// TIA Portal V20 export
DATA_BLOCK "ControlNodes"   // DB68
{ DB_Accessible_From_OPC_UA := 'FALSE' }
AUTHOR : ERsystem_FA2_DH. Kim
// stored: DBAccessibleFromOPCUA false, DBAccessibleFromWebserver false, MemoryReserve 100, Namespace Unit1.Em7
   VAR
      em { ExternalAccessible := 'False'; ExternalVisible := 'False'; ExternalWritable := 'False'} : "LAF_typeEmControlNode";
      cm { ExternalAccessible := 'False'; ExternalVisible := 'False'; ExternalWritable := 'False'} : Struct
         interlock : Struct
            sepaClampnCutterAxisX : "LER_typeAxisInterlock";
            sepaClampnCutterAxisZ : "LER_typeAxisInterlock";
            sepaGripperAxisX : "LER_typeAxisInterlock";
            sepaGripperAxisZ : "LER_typeAxisInterlock";
            sepaGripperAxisC : "LER_typeAxisInterlock";
            jrWinderRearAxisY : "LER_typeAxisInterlock";
            jrWinderFrontAxisY : "LER_typeAxisInterlock";
            jrWinderAxisB : "LER_typeAxisInterlock";
            jrPusherAxisZ : "LER_typeAxisInterlock";
            sepaCutterUpDown : "LER_typeTwoWayActInterlock";
            sepaClampTopUpDown : "LER_typeTwoWayActInterlock";
            sepaClampBottomUpDown : "LER_typeTwoWayActInterlock";
            stackGripperOpenClose : "LER_typeTwoWayActInterlock";
            stackGripperFwdBwd : "LER_typeTwoWayActInterlock";
            jrWinderClampTopRearUpDown : "LER_typeTwoWayActInterlock";
            jrWinderClampBtmRearUpDown : "LER_typeTwoWayActInterlock";
            jrWinderClampTopFrontUpDown : "LER_typeTwoWayActInterlock";
            jrWinderClampBtmFrontUpDown : "LER_typeTwoWayActInterlock";
            pusherRollerFwdBwd : "LER_typeTwoWayActInterlock";
         END_STRUCT;
         Command : Struct
            sepaClampnCutterAxisX : "LER_typeAxisCommand";
            sepaClampnCutterAxisZ : "LER_typeAxisCommand";
            sepaGripperAxisX : "LER_typeAxisCommand";
            sepaGripperAxisZ : "LER_typeAxisCommand";
            sepaGripperAxisC : "LER_typeAxisCommand";
            jrWinderRearAxisY : "LER_typeAxisCommand";
            jrWinderFrontAxisY : "LER_typeAxisCommand";
            jrWinderAxisB : "LER_typeAxisCommand";
            jrPusherAxisZ { S7_SetPoint := 'True'} : "LER_typeAxisCommand";
         END_STRUCT;
         softCam : "Unit1.type_emRelations_em7_SoftCam";
         brakeTest : Struct
            sepaClampnCutterAxisZ : "LER_typeBrakeTestEmControlNoeds";
            sepaGripperAxisZ : "LER_typeBrakeTestEmControlNoeds";
            jrPusherAxisZ : "LER_typeBrakeTestEmControlNoeds";
         END_STRUCT;
         calculateCam : Struct
            sepaClampnCutterAxisX : Struct
               execute : Bool;
               done : Bool;
               busy : Bool;
               error : Bool;
               errorID : DWord;
            END_STRUCT;
            sepaClampnCutterAxisZ : Struct
               execute : Bool;
               done : Bool;
               busy : Bool;
               error : Bool;
               errorID : DWord;
            END_STRUCT;
            jrPusherAxisZ : Struct
               execute : Bool;
               done : Bool;
               busy : Bool;
               error : Bool;
               errorID : DWord;
            END_STRUCT;
         END_STRUCT;
         CamIn : Struct
            sepaClampnCutterAxisX : Struct
               execute : Bool := false;
               MasterOffset : LReal := 0.0;
               SlaveOffset : LReal := 0.0;
               MasterScaling : LReal := 1.0;
               SlaveScaling : LReal := 1.0;
               MasterSyncPosition : LReal := 0.0;
               SyncProfileReference : DInt := 2;
               MasterStartDistance : LReal := 0.0;
               Velocity : LReal := -1.0;
               Acceleration : LReal := -1.0;
               Deceleration : LReal := -1.0;
               Jerk : LReal := -1.0;
               ApplicationMode : DInt := 2;
               SyncDirection : DInt := 3;
               StartSync : Bool;
               InSync : Bool;
               Busy : Bool;
               CommandAborted : Bool;
               Error : Bool;
               ErrorId : Word;
               EndOfProfile : Bool;
            END_STRUCT;
            sepaClampnCutterAxisZ : Struct
               execute : Bool := false;
               MasterOffset : LReal := 0.0;
               SlaveOffset : LReal := 0.0;
               MasterScaling : LReal := 1.0;
               SlaveScaling : LReal := 1.0;
               MasterSyncPosition : LReal := 0.0;
               SyncProfileReference : DInt := 2;
               MasterStartDistance : LReal := 0.0;
               Velocity : LReal := -1.0;
               Acceleration : LReal := -1.0;
               Deceleration : LReal := -1.0;
               Jerk : LReal := -1.0;
               ApplicationMode : DInt := 2;
               SyncDirection : DInt := 3;
               StartSync : Bool;
               InSync : Bool;
               Busy : Bool;
               CommandAborted : Bool;
               Error : Bool;
               ErrorId : Word;
               EndOfProfile : Bool;
            END_STRUCT;
            jrPusherAxisZ : Struct
               execute : Bool := false;
               MasterOffset : LReal := 0.0;
               SlaveOffset : LReal := 0.0;
               MasterScaling : LReal := 1.0;
               SlaveScaling : LReal := 1.0;
               MasterSyncPosition : LReal := 0.0;
               SyncProfileReference : DInt := 2;
               MasterStartDistance : LReal := 0.0;
               Velocity : LReal := -1.0;
               Acceleration : LReal := -1.0;
               Deceleration : LReal := -1.0;
               Jerk : LReal := -1.0;
               ApplicationMode : DInt := 2;
               SyncDirection : DInt := 3;
               StartSync : Bool;
               InSync : Bool;
               Busy : Bool;
               CommandAborted : Bool;
               Error : Bool;
               ErrorId : Word;
               EndOfProfile : Bool;
            END_STRUCT;
         END_STRUCT;
         CamUse : Struct
            CamUse : Bool;
         END_STRUCT;
      END_STRUCT;
      sepaClamp : Struct
         jobs : "LAF_typeJobs";
         sequence { S7_SetPoint := 'True'} : "LAF_typeSequence";
         "step" { S7_SetPoint := 'True'} : "LER_typeStep";
         jobInterface : Struct
            homeJob1 { ExternalAccessible := 'False'; ExternalVisible := 'False'; ExternalWritable := 'False'} : "LER_typeJobInterface";
            gripReadyJob2 { ExternalAccessible := 'False'; ExternalVisible := 'False'; ExternalWritable := 'False'; S7_SetPoint := 'True'} : "LER_typeJobInterface";
            clampAndCuttingJob3 { ExternalAccessible := 'False'; ExternalVisible := 'False'; ExternalWritable := 'False'; S7_SetPoint := 'True'} : "LER_typeJobInterface";
            winderMoveJob4 { ExternalAccessible := 'False'; ExternalVisible := 'False'; ExternalWritable := 'False'; S7_SetPoint := 'True'} : "LER_typeJobInterface";
            sepaWindingJob5 { ExternalAccessible := 'False'; ExternalVisible := 'False'; ExternalWritable := 'False'; S7_SetPoint := 'True'} : "LER_typeJobInterface";
            returnJob6 { ExternalAccessible := 'False'; ExternalVisible := 'False'; ExternalWritable := 'False'; S7_SetPoint := 'True'} : "LER_typeJobInterface";
            unloadCamJob10 { S7_SetPoint := 'True'} : "LER_typeJobInterface";
            unloadStopSyncJob11 { S7_SetPoint := 'True'} : "LER_typeJobInterface";
            unloadReturnJob12 { S7_SetPoint := 'True'} : "LER_typeJobInterface";
         END_STRUCT;
         preOperationCheck : Struct
            partNoDetect : Bool;
            partDetect : Bool;
            Bool3 : Bool;
            Bool4 : Bool;
            Bool5 : Bool;
            Bool6 : Bool;
            Bool7 : Bool;
            Bool8 : Bool;
            Bool9 : Bool;
            Bool10 : Bool;
            Bool11 : Bool;
            Bool12 : Bool;
            Bool13 : Bool;
            Bool14 : Bool;
            Bool15 : Bool;
            Bool16 : Bool;
            Bool17 : Bool;
            Bool18 : Bool;
            Bool19 : Bool;
            Bool20 : Bool;
         END_STRUCT;
      END_STRUCT;
      sepaGripper : Struct
         jobs : "LAF_typeJobs";
         sequence { S7_SetPoint := 'True'} : "LAF_typeSequence";
         "step" { S7_SetPoint := 'True'} : "LER_typeStep";
         jobInterface : Struct
            homeJob1 { ExternalAccessible := 'False'; ExternalVisible := 'False'; ExternalWritable := 'False'; S7_SetPoint := 'True'} : "LER_typeJobInterface";
            loadJob2 { ExternalAccessible := 'False'; ExternalVisible := 'False'; ExternalWritable := 'False'; S7_SetPoint := 'True'} : "LER_typeJobInterface";
            unloadJob3 { ExternalAccessible := 'False'; ExternalVisible := 'False'; ExternalWritable := 'False'; S7_SetPoint := 'True'} : "LER_typeJobInterface";
            reLoadJob4 { ExternalAccessible := 'False'; ExternalVisible := 'False'; ExternalWritable := 'False'; S7_SetPoint := 'True'} : "LER_typeJobInterface";
            reUnloadJob5 { ExternalAccessible := 'False'; ExternalVisible := 'False'; ExternalWritable := 'False'; S7_SetPoint := 'True'} : "LER_typeJobInterface";
            LoadToStackTableJob12 { S7_SetPoint := 'True'} : "LER_typeJobInterface";
            UnLoadToJRWinderJob13 { S7_SetPoint := 'True'} : "LER_typeJobInterface";
            LoadToJRWinderJob15 { S7_SetPoint := 'True'} : "LER_typeJobInterface";
            UnLoadToInspectionJob17 { S7_SetPoint := 'True'} : "LER_typeJobInterface";
            ReturnJob18 { S7_SetPoint := 'True'} : "LER_typeJobInterface";
         END_STRUCT;
         preOperationCheck : Struct
            partNoDetect1 : Bool;
            partDetect1 : Bool;
            partNoDetect2 : Bool;
            partDetect2 : Bool;
            partNoDetect1_Cam : Bool;
            partDetect1_Cam : Bool;
            partDetect2_Cam : Bool;
            partNoDetect2_Cam : Bool;
            partDetect3_Cam : Bool;
            partNoDetect3_Cam : Bool;
            Bool11 : Bool;
            Bool12 : Bool;
            Bool13 : Bool;
            Bool14 : Bool;
            Bool15 : Bool;
            Bool16 : Bool;
            Bool17 : Bool;
            Bool18 : Bool;
            Bool19 : Bool;
            Bool20 : Bool;
         END_STRUCT;
      END_STRUCT;
      jellyRollWinder : Struct
         jobs : "LAF_typeJobs";
         sequence { S7_SetPoint := 'True'} : "LAF_typeSequence";
         "step" { S7_SetPoint := 'True'} : "LER_typeStep";
         jobInterface : Struct
            homeJob1 { ExternalAccessible := 'False'; ExternalVisible := 'False'; ExternalWritable := 'False'; S7_SetPoint := 'True'} : "LER_typeJobInterface";
            loadJob2 { ExternalAccessible := 'False'; ExternalVisible := 'False'; ExternalWritable := 'False'; S7_SetPoint := 'True'} : "LER_typeJobInterface";
            winding1Job3 { ExternalAccessible := 'False'; ExternalVisible := 'False'; ExternalWritable := 'False'; S7_SetPoint := 'True'} : "LER_typeJobInterface";
            pusherReadyJob4 { ExternalAccessible := 'False'; ExternalVisible := 'False'; ExternalWritable := 'False'; S7_SetPoint := 'True'} : "LER_typeJobInterface";
            winding2Job5 { ExternalAccessible := 'False'; ExternalVisible := 'False'; ExternalWritable := 'False'; S7_SetPoint := 'True'} : "LER_typeJobInterface";
            unloadJob6 { ExternalAccessible := 'False'; ExternalVisible := 'False'; ExternalWritable := 'False'; S7_SetPoint := 'True'} : "LER_typeJobInterface";
            camWinding1stJob10 { S7_SetPoint := 'True'} : "LER_typeJobInterface";
            camPusherReadyJob11 { S7_SetPoint := 'True'} : "LER_typeJobInterface";
            camCamStartSyncJob12 { S7_SetPoint := 'True'} : "LER_typeJobInterface";
            camWinding2ndJob13 { S7_SetPoint := 'True'} : "LER_typeJobInterface";
            camStopSyncJob14 { S7_SetPoint := 'True'} : "LER_typeJobInterface";
         END_STRUCT;
         preOperationCheck : Struct
            partNoDetect : Bool;
            partDetect : Bool;
            winding1 : Bool;
            pusherReady : Bool;
            winding2 : Bool;
            Bool6 : Bool;
            Bool7 : Bool;
            Bool8 : Bool;
            Bool9 : Bool;
            Bool10 : Bool;
            Bool11 : Bool;
            Bool12 : Bool;
            Bool13 : Bool;
            Bool14 : Bool;
            Bool15 : Bool;
            Bool16 : Bool;
            Bool17 : Bool;
            Bool18 : Bool;
            Bool19 : Bool;
            Bool20 : Bool;
         END_STRUCT;
      END_STRUCT;
      inspectionInterface : Struct
         BA060 : Struct
            null : Bool;
         END_STRUCT;
      END_STRUCT;
      emRelations : Struct
         em4 : Struct
            softCam : "Unit1.type_emRelations_em4_SoftCam";
            cmStatus : Struct
               null : Bool;
            END_STRUCT;
         END_STRUCT;
         em6 : Struct
            softCam : "Unit1.type_emRelations_em6_SoftCam";
            cmStatus : Struct
               GapPadUpDown : "LBC_typeTwoWayActuatorControlNodeMonitoring";
            END_STRUCT;
         END_STRUCT;
      END_STRUCT;
      motionRelations : Struct
         commands : Struct
            unloadGripComplete : Bool;
            unloadClampLockComplete : Bool;
            unloadClampCuttingComplete : Bool;
            unloadJobComplete : Bool;
         END_STRUCT;
         monitoring : Struct
            stackComplete : Bool;
            stackUpComplete : Bool;
            stackUngripComplete : Bool;
            stackGripComplete : Bool;
         END_STRUCT;
         Config : Struct
            Null : Bool;
         END_STRUCT;
      END_STRUCT;
      cmSepaClampDetectSensor { ExternalAccessible := 'False'; ExternalVisible := 'False'; ExternalWritable := 'False'} : "LBC_typeDigitalSignalControlNode";
      cmSepaGripperDetectSensor { ExternalAccessible := 'False'; ExternalVisible := 'False'; ExternalWritable := 'False'} : "LBC_typeDigitalSignalControlNode";
      cmJRWinderDetectSensor { ExternalAccessible := 'False'; ExternalVisible := 'False'; ExternalWritable := 'False'} : "LBC_typeDigitalSignalControlNode";
      cmSepaClampSafetyPinDetectSensor { ExternalAccessible := 'False'; ExternalVisible := 'False'; ExternalWritable := 'False'} : "LBC_typeDigitalSignalControlNode";
      cmSepaGripperSafetyPinDetectSensor { ExternalAccessible := 'False'; ExternalVisible := 'False'; ExternalWritable := 'False'} : "LBC_typeDigitalSignalControlNode";
      cmSepaClampnCutterAxisX { ExternalAccessible := 'False'; ExternalVisible := 'False'; ExternalWritable := 'False'} : "LBC_typeAxis64PosControlNode";
      cmSepaClampnCutterAxisZ { ExternalAccessible := 'False'; ExternalVisible := 'False'; ExternalWritable := 'False'} : "LBC_typeAxis64PosControlNode";
      cmSepaGripperAxisX { ExternalAccessible := 'False'; ExternalVisible := 'False'; ExternalWritable := 'False'} : "LBC_typeAxis64PosControlNode";
      cmSepaGripperAxisZ { ExternalAccessible := 'False'; ExternalVisible := 'False'; ExternalWritable := 'False'} : "LBC_typeAxis64PosControlNode";
      cmSepaGripperAxisC { ExternalAccessible := 'False'; ExternalVisible := 'False'; ExternalWritable := 'False'} : "LBC_typeAxis64PosControlNode";
      cmJRWinderRearAxisY { ExternalAccessible := 'False'; ExternalVisible := 'False'; ExternalWritable := 'False'} : "LBC_typeAxis64PosControlNode";
      cmJRWinderFrontAxisY { ExternalAccessible := 'False'; ExternalVisible := 'False'; ExternalWritable := 'False'} : "LBC_typeAxis64PosControlNode";
      cmJRWinderAxisB { ExternalAccessible := 'False'; ExternalVisible := 'False'; ExternalWritable := 'False'} : "LBC_typeAxis64PosControlNode";
      cmJRPusherAxisZ { ExternalAccessible := 'False'; ExternalVisible := 'False'; ExternalWritable := 'False'} : "LBC_typeAxis64PosControlNode";
      cmSepaCutterUpDown { ExternalAccessible := 'False'; ExternalVisible := 'False'; ExternalWritable := 'False'} : "LBC_typeTwoWayActuatorControlNode";
      cmSepaClampTopUpDown { ExternalAccessible := 'False'; ExternalVisible := 'False'; ExternalWritable := 'False'} : "LBC_typeTwoWayActuatorControlNode";
      cmSepaClampBottomUpDown { ExternalAccessible := 'False'; ExternalVisible := 'False'; ExternalWritable := 'False'} : "LBC_typeTwoWayActuatorControlNode";
      cmStackGripperOpenClose { ExternalAccessible := 'False'; ExternalVisible := 'False'; ExternalWritable := 'False'} : "LBC_typeTwoWayActuatorControlNode";
      cmStackGripperFwdBwd { ExternalAccessible := 'False'; ExternalVisible := 'False'; ExternalWritable := 'False'} : "LBC_typeTwoWayActuatorControlNode";
      cmJRWinderClampTopRearUpDown { ExternalAccessible := 'False'; ExternalVisible := 'False'; ExternalWritable := 'False'} : "LBC_typeTwoWayActuatorControlNode";
      cmJRWinderClampBtmRearUpDown { ExternalAccessible := 'False'; ExternalVisible := 'False'; ExternalWritable := 'False'} : "LBC_typeTwoWayActuatorControlNode";
      cmJRWinderClampTopFrontUpDown { ExternalAccessible := 'False'; ExternalVisible := 'False'; ExternalWritable := 'False'} : "LBC_typeTwoWayActuatorControlNode";
      cmJRWinderClampBtmFrontUpDown { ExternalAccessible := 'False'; ExternalVisible := 'False'; ExternalWritable := 'False'} : "LBC_typeTwoWayActuatorControlNode";
      cmPusherRollerFwdBwd { ExternalAccessible := 'False'; ExternalVisible := 'False'; ExternalWritable := 'False'} : "LBC_typeTwoWayActuatorControlNode";
      cmHotWireCutter { ExternalAccessible := 'False'; ExternalVisible := 'False'; ExternalWritable := 'False'} : "LER_typeHotWireCutterControlNode";
   END_VAR
BEGIN
   em.commands.enable := FALSE;
   em.commands.acknowledge := FALSE;
   em.commands.disableAlarms := FALSE;
   em.commands.activateSimulation := FALSE;
   em.commands.home := FALSE;
   em.commands.moveToInitialPosition := FALSE;
   em.commands.directModeControl.current := 2;
   em.commands.directModeControl.production := FALSE;
   em.commands.directModeControl.maintenance := TRUE;
   em.commands.directModeControl.manual := FALSE;
   em.commands.directModeControl.nomode := FALSE;
   em.commands.directModeControl.sleep := FALSE;
   em.commands.directModeControl.deepsleep := FALSE;
   em.commands.directModeControl.userMode04 := FALSE;
   em.commands.directModeControl.userMode05 := FALSE;
   em.commands.directModeControl.userMode06 := FALSE;
   em.commands.directModeControl.userMode07 := FALSE;
   em.commands.directModeControl.userMode08 := FALSE;
   em.commands.directModeControl.userMode09 := FALSE;
   em.commands.directModeControl.userMode10 := FALSE;
   em.commands.directModeControl.userMode11 := FALSE;
   em.commands.directModeControl.userMode12 := FALSE;
   em.commands.directModeControl.userMode13 := FALSE;
   em.commands.directStateControl.current := 2;
   em.commands.directStateControl.clearing := FALSE;
   em.commands.directStateControl.stopped := TRUE;
   em.commands.directStateControl.starting := FALSE;
   em.commands.directStateControl.idle := FALSE;
   em.commands.directStateControl.suspended := FALSE;
   em.commands.directStateControl.execute := FALSE;
   em.commands.directStateControl.stopping := FALSE;
   em.commands.directStateControl.aborting := FALSE;
   em.commands.directStateControl.aborted := FALSE;
   em.commands.directStateControl.holding := FALSE;
   em.commands.directStateControl.held := FALSE;
   em.commands.directStateControl.unholding := FALSE;
   em.commands.directStateControl.suspending := FALSE;
   em.commands.directStateControl.unsuspending := FALSE;
   em.commands.directStateControl.resetting := FALSE;
   em.commands.directStateControl.completing := FALSE;
   em.commands.directStateControl.complete := FALSE;
   em.status.enabled := FALSE;
   em.status.acknowledgeActive := FALSE;
   em.status.alarmsDisabled := FALSE;
   em.status.simulationActive := FALSE;
   em.status.safetyReleased := TRUE;
   em.status.initialized := FALSE;
   em.status.homed := FALSE;
   em.status.safeState := FALSE;
   em.status.stateComplete := TRUE;
   // sepaClamp."step".action1[101] : Step[101] : JOB[1] Condition
   // sepaClamp."step".action1[110] : Step[110] : Cutter Up
   // sepaClamp."step".action1[120] : Step[120] : Cutter Heater Off
   // sepaClamp."step".action1[130] : Step[130] : Clamp Close
   // sepaClamp."step".action1[180] : Step[180] : Clamp X,Z-Axis Wait Pos
   // sepaClamp."step".action1[190] : Step[190] : Job[1] Step End
   // sepaClamp."step".action1[201] : Step[201] : JOB[2] Condition
   // sepaClamp."step".action1[210] : Step[210] : Clamp X,Z-Axis Load Pos
   // sepaClamp."step".action1[220] : Step[220] : Clamp Open
   // sepaClamp."step".action1[221] : Step[221] : Sepa Clamp → Sepa Gripper [Loading Ready]
   // sepaClamp."step".action1[230] : Step[230] : Clamp Close
   // sepaClamp."step".action1[240] : Step[240] : Cutter Heater On
   // sepaClamp."step".action1[250] : Step[250] : Cutter Down
   // sepaClamp."step".action1[251] : Step[251] : Cutter Up
   // sepaClamp."step".action1[260] : Step[260] : Cutter Heater Off
   // sepaClamp."step".action1[280] : Step[280] : Clamp X,Z-Axis Winding Ready Pos
   // sepaClamp."step".action1[290] : Step[290] : Job[2] Step End
   // sepaClamp."step".action1[301] : Step[301] : JOB[3] Condition
   // sepaClamp."step".action1[310] : Step[310] : Sepa Clamp → JR Winder [Unloading Ready]
   // sepaClamp."step".action1[320] : Step[320] : Clamp X-Axis Winding Move Pos
   // sepaClamp."step".action1[321] : Step[321] : Sepa Clamp → JR Winder [UnClamp Ready]
   // sepaClamp."step".action1[330] : Step[330] : Clamp Open
   // sepaClamp."step".action1[331] : Step[331] : Sepa Clamp → JR Winder [Unloading Done]
   // sepaClamp."step".action1[340] : Step[340] : Clamp Close
   // sepaClamp."step".action1[380] : Step[380] : Clamp X,Z-Axis Wait Pos
   // sepaClamp."step".action1[390] : Step[390] : Job[3] Step End
   // sepaClamp."step".action1[401] : Step[401] : JOB[4] Condition
   // sepaClamp."step".action1[410] : Step[410] : Clamp X-Axis Winder Pos
   // sepaClamp."step".action1[411] : Step[411] : Clamp Z-Axis Winder Pos
   // sepaClamp."step".action1[490] : Step[490] : Job[4] Step End
   // sepaClamp."step".action1[501] : Step[501] : Job[5] Condition
   // sepaClamp."step".action1[510] : Step[510] : CamIn Config
   // sepaClamp."step".action1[511] : Step[511] : Clamp X-Axis CamIn
   // sepaClamp."step".action1[520] : Step[520] : Check Clamp X-Axis WinderDone Pos
   // sepaClamp."step".action1[521] : Step[521] : Clamp X-Axis Halt
   // sepaClamp."step".action1[530] : Step[530] : Clamp Open
   // sepaClamp."step".action1[590] : Step[590] : Job[5] Step End
   // sepaClamp."step".action1[601] : Step[601] : JOB[6] Condition
   // sepaClamp."step".action1[610] : Step[610] : Cutter Up
   // sepaClamp."step".action1[611] : Step[611] : Clamp Close
   // sepaClamp."step".action1[620] : Step[620] : Clamp Z-Axis WaitPos
   // sepaClamp."step".action1[630] : Step[630] : Clamp X-Axis WaitPos
   // sepaClamp."step".action1[690] : Step[690] : Job[6] Step End
   // sepaClamp."step".action1[1001] : Step[1001] : JOB[10] Condition
   // sepaClamp."step".action1[1010] : Step[1010] : Sepa Clamp X/Z Cam Calculate
   // sepaClamp."step".action1[1011] : Step[1011] : Sepa Clamp X/Z CamIn
   // sepaClamp."step".action1[1090] : Step[1090] : Job[10] Step End
   // sepaClamp."step".action1[1101] : Step[1101] : JOB[11] Condition
   // sepaClamp."step".action1[1110] : Step[1110] : Clamp Top Open
   // sepaClamp."step".action1[1120] : Step[1120] : Sepa Clamp Halt [Stop Sync]
   // sepaClamp."step".action1[1130] : Step[1130] : Clamp Top Close
   // sepaClamp."step".action1[1190] : Step[1190] : Job[11] Step End
   // sepaClamp."step".action1[1201] : Step[1201] : JOB[12] Condition
   // sepaClamp."step".action1[1210] : Step[1210] : Clamp X,Z-Axis Wait Pos
   // sepaClamp."step".action1[1290] : Step[1290] : Job[12] Step End
   // sepaClamp."step".transition1[101] : Step[101] : JOB[1] Condition
   // sepaClamp."step".transition1[110] : Step[110] : Cutter Up
   // sepaClamp."step".transition1[120] : Step[120] : Cutter Heater Off
   // sepaClamp."step".transition1[130] : Step[130] : Clamp Close
   // sepaClamp."step".transition1[180] : Step[180] : Clamp X,Z-Axis Wait Pos
   // sepaClamp."step".transition1[190] : Step[190] : Job[1] Step End
   // sepaClamp."step".transition1[201] : Step[201] : JOB[2] Condition
   // sepaClamp."step".transition1[210] : Step[210] : Clamp X,Z-Axis Load Pos
   // sepaClamp."step".transition1[220] : Step[220] : Clamp Open
   // sepaClamp."step".transition1[221] : Step[221] : Sepa Clamp → Sepa Gripper [Loading Ready]
   // sepaClamp."step".transition1[230] : Step[230] : Clamp Close
   // sepaClamp."step".transition1[240] : Step[240] : Cutter Heater On
   // sepaClamp."step".transition1[250] : Step[250] : Cutter Down
   // sepaClamp."step".transition1[251] : Step[251] : Cutter Up
   // sepaClamp."step".transition1[260] : Step[260] : Cutter Heater Off
   // sepaClamp."step".transition1[280] : Step[280] : Clamp X,Z-Axis Winding Ready Pos
   // sepaClamp."step".transition1[290] : Step[290] : Job[2] Step End
   // sepaClamp."step".transition1[301] : Step[301] : JOB[3] Condition
   // sepaClamp."step".transition1[310] : Step[310] : Sepa Clamp → JR Winder [Unloading Ready]
   // sepaClamp."step".transition1[320] : Step[320] : Clamp X-Axis Winding Move Pos
   // sepaClamp."step".transition1[321] : Step[321] : Sepa Clamp → JR Winder [UnClamp Ready]
   // sepaClamp."step".transition1[330] : Step[330] : Clamp Open
   // sepaClamp."step".transition1[331] : Step[331] : Sepa Clamp → JR Winder [Unloading Done]
   // sepaClamp."step".transition1[340] : Step[340] : Clamp Close
   // sepaClamp."step".transition1[380] : Step[380] : Clamp X,Z-Axis Wait Pos
   // sepaClamp."step".transition1[390] : Step[390] : Job[3] Step End
   // sepaClamp."step".transition1[401] : Step[401] : JOB[4] Condition
   // sepaClamp."step".transition1[410] : Step[410] : Clamp X-Axis Winder Pos
   // sepaClamp."step".transition1[411] : Step[411] : Clamp Z-Axis Winder Pos
   // sepaClamp."step".transition1[490] : Step[490] : Job[4] Step End
   // sepaClamp."step".transition1[501] : Step[501] : Job[5] Condition
   // sepaClamp."step".transition1[510] : Step[510] : CamIn Config
   // sepaClamp."step".transition1[511] : Step[511] : Clamp X-Axis CamIn
   // sepaClamp."step".transition1[520] : Step[520] : Check Clamp X-Axis WinderDone Pos
   // sepaClamp."step".transition1[521] : Step[521] : Clamp X-Axis Halt
   // sepaClamp."step".transition1[530] : Step[530] : Clamp Open
   // sepaClamp."step".transition1[590] : Step[590] : Job[5] Step End
   // sepaClamp."step".transition1[601] : Step[601] : JOB[6] Condition
   // sepaClamp."step".transition1[610] : Step[610] : Cutter Up
   // sepaClamp."step".transition1[611] : Step[611] : Clamp Close
   // sepaClamp."step".transition1[620] : Step[620] : Clamp Z-Axis WaitPos
   // sepaClamp."step".transition1[630] : Step[630] : Clamp X-Axis WaitPos
   // sepaClamp."step".transition1[690] : Step[690] : Job[6] Step End
   // sepaClamp."step".transition1[1001] : Step[1001] : JOB[10] Condition
   // sepaClamp."step".transition1[1010] : Step[1010] : Sepa Clamp X/Z Cam Calculate
   // sepaClamp."step".transition1[1011] : Step[1011] : Sepa Clamp X/Z CamIn
   // sepaClamp."step".transition1[1090] : Step[1090] : Job[10] Step End
   // sepaClamp."step".transition1[1101] : Step[1101] : JOB[11] Condition
   // sepaClamp."step".transition1[1110] : Step[1110] : Clamp Top Open
   // sepaClamp."step".transition1[1120] : Step[1120] : Sepa Clamp Halt [Stop Sync]
   // sepaClamp."step".transition1[1130] : Step[1130] : Clamp Top Close
   // sepaClamp."step".transition1[1190] : Step[1190] : Job[11] Step End
   // sepaClamp."step".transition1[1201] : Step[1201] : JOB[12] Condition
   // sepaClamp."step".transition1[1210] : Step[1210] : Clamp X,Z-Axis Wait Pos
   // sepaClamp."step".transition1[1290] : Step[1290] : Job[12] Step End
   // sepaGripper."step".action1[101] : Step[101] : JOB [Homing] Condition
   // sepaGripper."step".action1[110] : Step[110] : Gripper Open
   // sepaGripper."step".action1[120] : Step[120] : Gripper Backward
   // sepaGripper."step".action1[130] : Step[130] : Gripper X-Axis SepaTailPos
   // sepaGripper."step".action1[140] : Step[140] : Gripper X-Axis Turn Pos
   // sepaGripper."step".action1[141] : Step[141] : Gripper Z-Axis Turn Pos
   // sepaGripper."step".action1[150] : Step[150] : Gripper C-Axis Wait Pos
   // sepaGripper."step".action1[180] : Step[180] : Gripper X,Z-Axis Wait Pos
   // sepaGripper."step".action1[190] : Step[190] : Job[1] Step End
   // sepaGripper."step".action1[201] : Step[201] : JOB[2] Condition
   // sepaGripper."step".action1[210] : Step[210] : Gripper X,Z-Axis Load Pos
   // sepaGripper."step".action1[220] : Step[220] : Gripper Forward
   // sepaGripper."step".action1[230] : Step[230] : Gripper Close
   // sepaGripper."step".action1[231] : Step[231] : Sepa Gripper → Stack Table [Loading Ready]
   // sepaGripper."step".action1[240] : Step[240] : Gripper Backward
   // sepaGripper."step".action1[250] : Step[250] : Gripper X-Axis Sepa Tail Pos
   // sepaGripper."step".action1[251] : Step[251] : Gripper → Stack Table [Loading Done]
   // sepaGripper."step".action1[280] : Step[280] : Gripper X,Z-Axis Winding Ready Pos
   // sepaGripper."step".action1[290] : Step[290] : Job[2] Step End
   // sepaGripper."step".action1[301] : Step[301] : JOB[3] Condition
   // sepaGripper."step".action1[310] : Step[310] : Sepa Gripper → JR Winder [Unloading Ready]
   // sepaGripper."step".action1[320] : Step[320] : Gripper Open
   // sepaGripper."step".action1[330] : Step[330] : Gripper X-Axis Avoid Pos
   // sepaGripper."step".action1[390] : Step[390] : Job[3] Step End
   // sepaGripper."step".action1[401] : Step[401] : JOB[4] Condition
   // sepaGripper."step".action1[410] : Step[410] : Gripper X,Z-Axis Reload Pos
   // sepaGripper."step".action1[420] : Step[420] : Gripper Close
   // sepaGripper."step".action1[421] : Step[421] : Sepa Gripper → JR Winder [Loading Ready]
   // sepaGripper."step".action1[430] : Step[430] : Gripper X,Z-Axis Turn Pos
   // sepaGripper."step".action1[490] : Step[490] : Job[4] Step End
   // sepaGripper."step".action1[501] : Step[501] : JOB[5] Condition
   // sepaGripper."step".action1[510] : Step[510] : Sepa Gripper → Inspection [Unloading Ready]
   // sepaGripper."step".action1[520] : Step[520] : Gripper C-Axis Unload Pos
   // sepaGripper."step".action1[530] : Step[530] : Gripper X,Z-Axis Unload Pos
   // sepaGripper."step".action1[531] : Step[531] : Sepa Gripper → Inspection [Clamp Request]
   // sepaGripper."step".action1[540] : Step[540] : Gripper Open
   // sepaGripper."step".action1[550] : Step[550] : Gripper X,Z-Axis Turn Pos
   // sepaGripper."step".action1[580] : Step[580] : Gripper X,Z,C-Axis Wait Pos
   // sepaGripper."step".action1[581] : Step[581] : Sepa Gripper → Inspection [Unloading Done]
   // sepaGripper."step".action1[590] : Step[590] : Job[5] Step End
   // sepaGripper."step".action1[601] : Step[601] : JOB[6] Condition
   // sepaGripper."step".action1[610] : Step[610] : Gripper Z-Axis RePickUp Pos
   // sepaGripper."step".action1[611] : Step[611] : Gripper X-Axis Winder Pos
   // sepaGripper."step".action1[620] : Step[620] : Gripper Close
   // sepaGripper."step".action1[690] : Step[690] : Job[6] Step End
   // sepaGripper."step".action1[701] : Step[701] : JOB[7] Condition
   // sepaGripper."step".action1[710] : Step[710] : Gripper X-Axis Turn/Discharge Pos
   // sepaGripper."step".action1[720] : Step[720] : Gripper Z-Axis Turn Pos
   // sepaGripper."step".action1[730] : Step[730] : Gripper C-Axis OKDischarge Pos
   // sepaGripper."step".action1[740] : Step[740] : Gripper Z-Axis OKDischarge Pos
   // sepaGripper."step".action1[750] : Step[750] : Gripper X-Axis Avoid Pos
   // sepaGripper."step".action1[790] : Step[790] : Job[7] Step End
   // sepaGripper."step".action1[801] : Step[801] : JOB[8] Condition
   // sepaGripper."step".action1[810] : Step[810] : Gripper [Inspection Loader On] => Inspection
   // sepaGripper."step".action1[811] : Step[811] : Gripper X-Axis Ok DisCharge Pos
   // sepaGripper."step".action1[820] : Step[820] : Gripper [Inspection UnClamp Req] => Inspection
   // sepaGripper."step".action1[821] : Step[821] : Gripper Open
   // sepaGripper."step".action1[830] : Step[830] : Gripper [Inspection Avoid Req] => Inspection
   // sepaGripper."step".action1[831] : Step[831] : Gripper X-Axis Avoid Pos
   // sepaGripper."step".action1[890] : Step[890] : Job[8] Step End
   // sepaGripper."step".action1[901] : Step[901] : JOB[9] Condition
   // sepaGripper."step".action1[910] : Step[910] : Gripper X-Axis Turn/DisCharge Pos
   // sepaGripper."step".action1[920] : Step[920] : Gripper Z-Axis Turn Pos
   // sepaGripper."step".action1[930] : Step[930] : Gripper C-Axis Wait Pos
   // sepaGripper."step".action1[940] : Step[940] : Gripper X-Axis Wait Pos
   // sepaGripper."step".action1[950] : Step[950] : Gripper Z-Axis Wait Pos
   // sepaGripper."step".action1[990] : Step[990] : Job[9] Step End
   // sepaGripper."step".transition1[101] : Step[101] : JOB [Homing] Condition
   // sepaGripper."step".transition1[110] : Step[110] : Gripper Open
   // sepaGripper."step".transition1[120] : Step[120] : Gripper Backward
   // sepaGripper."step".transition1[130] : Step[130] : Gripper X-Axis SepaTailPos
   // sepaGripper."step".transition1[140] : Step[140] : Gripper X-Axis Turn Pos
   // sepaGripper."step".transition1[141] : Step[141] : Gripper Z-Axis Turn Pos
   // sepaGripper."step".transition1[150] : Step[150] : Gripper C-Axis Wait Pos
   // sepaGripper."step".transition1[180] : Step[180] : Gripper X,Z-Axis Wait Pos
   // sepaGripper."step".transition1[190] : Step[190] : Job[1] Step End
   // sepaGripper."step".transition1[201] : Step[201] : JOB[2] Condition
   // sepaGripper."step".transition1[210] : Step[210] : Gripper X,Z-Axis Load Pos
   // sepaGripper."step".transition1[220] : Step[220] : Gripper Forward
   // sepaGripper."step".transition1[230] : Step[230] : Gripper Close
   // sepaGripper."step".transition1[231] : Step[231] : Sepa Gripper → Stack Table [Loading Ready]
   // sepaGripper."step".transition1[240] : Step[240] : Gripper Backward
   // sepaGripper."step".transition1[250] : Step[250] : Gripper X-Axis Sepa Tail Pos
   // sepaGripper."step".transition1[251] : Step[251] : Gripper → Stack Table [Loading Done]
   // sepaGripper."step".transition1[280] : Step[280] : Gripper X,Z-Axis Winding Ready Pos
   // sepaGripper."step".transition1[290] : Step[290] : Job[2] Step End
   // sepaGripper."step".transition1[301] : Step[301] : JOB[3] Condition
   // sepaGripper."step".transition1[310] : Step[310] : Sepa Gripper → JR Winder [Unloading Ready]
   // sepaGripper."step".transition1[320] : Step[320] : Gripper Open
   // sepaGripper."step".transition1[330] : Step[330] : Gripper X-Axis Avoid Pos
   // sepaGripper."step".transition1[390] : Step[390] : Job[3] Step End
   // sepaGripper."step".transition1[401] : Step[401] : JOB[4] Condition
   // sepaGripper."step".transition1[410] : Step[410] : Gripper X,Z-Axis Reload Pos
   // sepaGripper."step".transition1[420] : Step[420] : Gripper Close
   // sepaGripper."step".transition1[421] : Step[421] : Sepa Gripper → JR Winder [Loading Ready]
   // sepaGripper."step".transition1[430] : Step[430] : Gripper X,Z-Axis Turn Pos
   // sepaGripper."step".transition1[490] : Step[490] : Job[4] Step End
   // sepaGripper."step".transition1[501] : Step[501] : JOB[5] Condition
   // sepaGripper."step".transition1[510] : Step[510] : Sepa Gripper → Inspection [Unloading Ready]
   // sepaGripper."step".transition1[520] : Step[520] : Gripper C-Axis Unload Pos
   // sepaGripper."step".transition1[530] : Step[530] : Gripper X,Z-Axis Unload Pos
   // sepaGripper."step".transition1[531] : Step[531] : Sepa Gripper → Inspection [Clamp Request]
   // sepaGripper."step".transition1[540] : Step[540] : Gripper Open
   // sepaGripper."step".transition1[550] : Step[550] : Gripper X,Z-Axis Turn Pos
   // sepaGripper."step".transition1[580] : Step[580] : Gripper X,Z,C-Axis Wait Pos
   // sepaGripper."step".transition1[581] : Step[581] : Sepa Gripper → Inspection [Unloading Done]
   // sepaGripper."step".transition1[590] : Step[590] : Job[5] Step End
   // sepaGripper."step".transition1[601] : Step[601] : JOB[6] Condition
   // sepaGripper."step".transition1[610] : Step[610] : Gripper Z-Axis RePickUp Pos
   // sepaGripper."step".transition1[611] : Step[611] : Gripper X-Axis Winder Pos
   // sepaGripper."step".transition1[620] : Step[620] : Gripper Close
   // sepaGripper."step".transition1[690] : Step[690] : Job[6] Step End
   // sepaGripper."step".transition1[701] : Step[701] : JOB[7] Condition
   // sepaGripper."step".transition1[710] : Step[710] : Gripper X-Axis Turn/Discharge Pos
   // sepaGripper."step".transition1[720] : Step[720] : Gripper Z-Axis Turn Pos
   // sepaGripper."step".transition1[730] : Step[730] : Gripper C-Axis OKDischarge Pos
   // sepaGripper."step".transition1[740] : Step[740] : Gripper Z-Axis OKDischarge Pos
   // sepaGripper."step".transition1[750] : Step[750] : Gripper X-Axis Avoid Pos
   // sepaGripper."step".transition1[790] : Step[790] : Job[7] Step End
   // sepaGripper."step".transition1[801] : Step[801] : JOB[8] Condition
   // sepaGripper."step".transition1[810] : Step[810] : Gripper [Inspection Loader On] => Inspection
   // sepaGripper."step".transition1[811] : Step[811] : Gripper X-Axis Ok DisCharge Pos
   // sepaGripper."step".transition1[820] : Step[820] : Gripper [Inspection UnClamp Req] => Inspection
   // sepaGripper."step".transition1[821] : Step[821] : Gripper Open
   // sepaGripper."step".transition1[830] : Step[830] : Gripper [Inspection Avoid Req] => Inspection
   // sepaGripper."step".transition1[831] : Step[831] : Gripper X-Axis Avoid Pos
   // sepaGripper."step".transition1[890] : Step[890] : Job[8] Step End
   // sepaGripper."step".transition1[901] : Step[901] : JOB[9] Condition
   // sepaGripper."step".transition1[910] : Step[910] : Gripper X-Axis Turn/DisCharge Pos
   // sepaGripper."step".transition1[920] : Step[920] : Gripper Z-Axis Turn Pos
   // sepaGripper."step".transition1[930] : Step[930] : Gripper C-Axis Wait Pos
   // sepaGripper."step".transition1[940] : Step[940] : Gripper X-Axis Wait Pos
   // sepaGripper."step".transition1[950] : Step[950] : Gripper Z-Axis Wait Pos
   // sepaGripper."step".transition1[990] : Step[990] : Job[9] Step End
   // jellyRollWinder."step".action1[101] : Step[101] : JOB[1] Condition
   // jellyRollWinder."step".action1[110] : Step[110] : Pusher Z-Axis Wait Pos
   // jellyRollWinder."step".action1[120] : Step[120]: Pusher Backward
   // jellyRollWinder."step".action1[130] : Step[130] : Winder Open
   // jellyRollWinder."step".action1[180] : Step[180] : Winder Y,B-Axis Wait Pos
   // jellyRollWinder."step".action1[190] : Step[190] : Job[1] Step End
   // jellyRollWinder."step".action1[201] : Step[201] : JOB[2] Condition
   // jellyRollWinder."step".action1[210] : Step[210] : Winder Y-Axis Grip Pos
   // jellyRollWinder."step".action1[220] : Step[220] : Winder Close
   // jellyRollWinder."step".action1[221] : Step[221] : Winder → Sepa Gripper [Loading Done]
   // jellyRollWinder."step".action1[290] : Step[290] : Job[2] Step End
   // jellyRollWinder."step".action1[301] : Step[301] : JOB[3] Condition
   // jellyRollWinder."step".action1[310] : Step[310] : Winder B-Axis Winding 1 Pos
   // jellyRollWinder."step".action1[390] : Step[390] : Job[3] Step End
   // jellyRollWinder."step".action1[401] : Step[401] : JOB[4] Condition
   // jellyRollWinder."step".action1[410] : Step[410] : Pusher Forward
   // jellyRollWinder."step".action1[420] : Step[420] : Pusher Z-Axis Work(=Down) Pos
   // jellyRollWinder."step".action1[421] : Step[421] : Winder → Sepa Clamp [Unclamp Request]
   // jellyRollWinder."step".action1[490] : Step[490] : Job[4] Step End
   // jellyRollWinder."step".action1[501] : Step[501] : JOB[5] Condition
   // jellyRollWinder."step".action1[510] : Step[510] : Winder B-Axis Winding 2 Vertical Pos, Pusher Vertical Pos
   // jellyRollWinder."step".action1[520] : Step[520] : Winder B-Axis Winding 2 Horizon Pos, Pusher Horizon Pos
   // jellyRollWinder."step".action1[590] : Step[590] : Job[5] Step End
   // jellyRollWinder."step".action1[601] : Step[601] : JOB[6] Condition
   // jellyRollWinder."step".action1[610] : Step[610] : Pusher Z-Axis Wait(=Up) Pos
   // jellyRollWinder."step".action1[620] : Step[620] : Pusehr Backward
   // jellyRollWinder."step".action1[621] : Step[621] : Winder → Sepa Gripper [Unloading Request]
   // jellyRollWinder."step".action1[630] : Step[630] : Winder Open
   // jellyRollWinder."step".action1[680] : Step[680] : Winder Y,B-Axis Wait Pos
   // jellyRollWinder."step".action1[690] : Step[690] : Job[6] Step End
   // jellyRollWinder."step".action1[701] : Step[701] : JOB[7] Condition
   // jellyRollWinder."step".action1[710] : Step[710] : Pusehr Z-axis Wait Pos
   // jellyRollWinder."step".action1[720] : Step[720] : Pusher Backward
   // jellyRollWinder."step".action1[730] : Step[730] : Clamp Open
   // jellyRollWinder."step".action1[740] : Step[740] : Winder Y-Axis Wait Pos
   // jellyRollWinder."step".action1[750] : Step[750] : Winder B-Axis Wait Pos
   // jellyRollWinder."step".action1[790] : Step[790] : Job[7] Step End
   // jellyRollWinder."step".action1[1001] : Step[1001] : JOB[10] Condition
   // jellyRollWinder."step".action1[1010] : Step[1010] : Winder B-Axis 1st Widning Pos
   // jellyRollWinder."step".action1[1090] : Step[1090] : Job[10] Step End
   // jellyRollWinder."step".action1[1101] : Step[1101] : JOB[11] Condition
   // jellyRollWinder."step".action1[1110] : Step[1110] : Pusher Forward
   // jellyRollWinder."step".action1[1120] : Step[1120] : Pusher Z-Axis Work(=Down) Pos
   // jellyRollWinder."step".action1[1190] : Step[1190] : Job[11] Step End
   // jellyRollWinder."step".action1[1201] : Step[1201] : JOB[12] Condition
   // jellyRollWinder."step".action1[1210] : Step[1210] : Pusher Z-Axis Cam Calculate
   // jellyRollWinder."step".action1[1211] : Step[1211] : Pusher Z-Axis CamIn [InSync]
   // jellyRollWinder."step".action1[1290] : Step[1290] : Job[12] Step End
   // jellyRollWinder."step".action1[1301] : Step[1301] : JOB[13] Condition
   // jellyRollWinder."step".action1[1310] : Step[1310] : Winder B-Axis 2nd Widning Pos
   // jellyRollWinder."step".action1[1390] : Step[1390] : Job[13] Step End
   // jellyRollWinder."step".action1[1401] : Step[1401] : JOB[14] Condition
   // jellyRollWinder."step".action1[1410] : Step[1410] : Pusher Halt [Stop Sync]
   // jellyRollWinder."step".action1[1490] : Step[1490] : Job[14] Step End
   // jellyRollWinder."step".transition1[101] : Step[101] : JOB[1] Condition
   // jellyRollWinder."step".transition1[110] : Step[110] : Pusher Z-Axis Wait Pos
   // jellyRollWinder."step".transition1[120] : Step[120]: Pusher Backward
   // jellyRollWinder."step".transition1[130] : Step[130] : Winder Open
   // jellyRollWinder."step".transition1[180] : Step[180] : Winder Y,B-Axis Wait Pos
   // jellyRollWinder."step".transition1[190] : Step[190] : Job[1] Step End
   // jellyRollWinder."step".transition1[201] : Step[201] : JOB[2] Condition
   // jellyRollWinder."step".transition1[210] : Step[210] : Winder Y-Axis Grip Pos
   // jellyRollWinder."step".transition1[220] : Step[220] : Winder Close
   // jellyRollWinder."step".transition1[221] : Step[221] : Winder → Sepa Gripper [Loading Done]
   // jellyRollWinder."step".transition1[290] : Step[290] : Job[2] Step End
   // jellyRollWinder."step".transition1[301] : Step[301] : JOB[3] Condition
   // jellyRollWinder."step".transition1[310] : Step[310] : Winder B-Axis Winding 1 Pos
   // jellyRollWinder."step".transition1[390] : Step[390] : Job[3] Step End
   // jellyRollWinder."step".transition1[401] : Step[401] : JOB[4] Condition
   // jellyRollWinder."step".transition1[410] : Step[410] : Pusher Forward
   // jellyRollWinder."step".transition1[420] : Step[420] : Pusher Z-Axis Work(=Down) Pos
   // jellyRollWinder."step".transition1[421] : Step[421] : Winder → Sepa Clamp [Unclamp Request]
   // jellyRollWinder."step".transition1[490] : Step[490] : Job[4] Step End
   // jellyRollWinder."step".transition1[501] : Step[501] : JOB[5] Condition
   // jellyRollWinder."step".transition1[510] : Step[510] : Winder B-Axis Winding 2 Vertical Pos, Pusher Vertical Pos
   // jellyRollWinder."step".transition1[520] : Step[520] : Winder B-Axis Winding 2 Horizon Pos, Pusher Horizon Pos
   // jellyRollWinder."step".transition1[590] : Step[590] : Job[5] Step End
   // jellyRollWinder."step".transition1[601] : Step[601] : JOB[6] Condition
   // jellyRollWinder."step".transition1[610] : Step[610] : Pusher Z-Axis Wait(=Up) Pos
   // jellyRollWinder."step".transition1[620] : Step[620] : Pusehr Backward
   // jellyRollWinder."step".transition1[621] : Step[621] : Winder → Sepa Gripper [Unloading Request]
   // jellyRollWinder."step".transition1[630] : Step[630] : Winder Open
   // jellyRollWinder."step".transition1[680] : Step[680] : Winder Y,B-Axis Wait Pos
   // jellyRollWinder."step".transition1[690] : Step[690] : Job[6] Step End
   // jellyRollWinder."step".transition1[701] : Step[701] : JOB[7] Condition
   // jellyRollWinder."step".transition1[710] : Step[710] : Pusehr Z-axis Wait Pos
   // jellyRollWinder."step".transition1[720] : Step[720] : Pusher Backward
   // jellyRollWinder."step".transition1[730] : Step[730] : Clamp Open
   // jellyRollWinder."step".transition1[740] : Step[740] : Winder Y-Axis Wait Pos
   // jellyRollWinder."step".transition1[750] : Step[750] : Winder B-Axis Wait Pos
   // jellyRollWinder."step".transition1[790] : Step[790] : Job[7] Step End
   // jellyRollWinder."step".transition1[1001] : Step[1001] : JOB[10] Condition
   // jellyRollWinder."step".transition1[1010] : Step[1010] : Winder B-Axis 1st Widning Pos
   // jellyRollWinder."step".transition1[1090] : Step[1090] : Job[10] Step End
   // jellyRollWinder."step".transition1[1101] : Step[1101] : JOB[11] Condition
   // jellyRollWinder."step".transition1[1110] : Step[1110] : Pusher Forward
   // jellyRollWinder."step".transition1[1120] : Step[1120] : Pusher Z-Axis Work(=Down) Pos
   // jellyRollWinder."step".transition1[1190] : Step[1190] : Job[11] Step End
   // jellyRollWinder."step".transition1[1201] : Step[1201] : JOB[12] Condition
   // jellyRollWinder."step".transition1[1210] : Step[1210] : Pusher Z-Axis Cam Calculate
   // jellyRollWinder."step".transition1[1211] : Step[1211] : Pusher Z-Axis CamIn [InSync]
   // jellyRollWinder."step".transition1[1290] : Step[1290] : Job[12] Step End
   // jellyRollWinder."step".transition1[1301] : Step[1301] : JOB[13] Condition
   // jellyRollWinder."step".transition1[1310] : Step[1310] : Winder B-Axis 2nd Widning Pos
   // jellyRollWinder."step".transition1[1390] : Step[1390] : Job[13] Step End
   // jellyRollWinder."step".transition1[1401] : Step[1401] : JOB[14] Condition
   // jellyRollWinder."step".transition1[1410] : Step[1410] : Pusher Halt [Stop Sync]
   // jellyRollWinder."step".transition1[1490] : Step[1490] : Job[14] Step End
   cmSepaClampnCutterAxisX.commandConfiguration.power.startMode := 1;
   cmSepaClampnCutterAxisX.commandConfiguration.power.stopMode := 0;
   cmSepaClampnCutterAxisX.commandConfiguration.power.syncMotionSimulation := FALSE;
   cmSepaClampnCutterAxisX.commandConfiguration.power.syncMotionSimulationExtendedMode := -1;
   cmSepaClampnCutterAxisX.commandConfiguration.jog.velocity := 0.0;
   cmSepaClampnCutterAxisX.commandConfiguration.jog.acceleration := -1.0;
   cmSepaClampnCutterAxisX.commandConfiguration.jog.deceleration := -1.0;
   cmSepaClampnCutterAxisX.commandConfiguration.jog.jerk := -1.0;
   cmSepaClampnCutterAxisX.commandConfiguration.jog.positionControlled := TRUE;
   cmSepaClampnCutterAxisX.commandConfiguration.jog.increment := 0.0;
   cmSepaClampnCutterAxisX.commandConfiguration.jog.mode := 0;
   cmSepaClampnCutterAxisX.commandConfiguration.moveVelocity.velocity := 0.0;
   cmSepaClampnCutterAxisX.commandConfiguration.moveVelocity.acceleration := -1.0;
   cmSepaClampnCutterAxisX.commandConfiguration.moveVelocity.deceleration := -1.0;
   cmSepaClampnCutterAxisX.commandConfiguration.moveVelocity.jerk := -1.0;
   cmSepaClampnCutterAxisX.commandConfiguration.moveVelocity.direction := 0;
   cmSepaClampnCutterAxisX.commandConfiguration.moveVelocity.positionControlled := TRUE;
   cmSepaClampnCutterAxisX.commandConfiguration.moveVelocity.velocityChangeOnTheFly := FALSE;
   cmSepaClampnCutterAxisX.commandConfiguration.stop.deceleration := -1.0;
   cmSepaClampnCutterAxisX.commandConfiguration.stop.jerk := -1.0;
   cmSepaClampnCutterAxisX.commandConfiguration.stop.abortAcceleration := FALSE;
   cmSepaClampnCutterAxisX.commandConfiguration.fastStop.deceleration := -1.0;
   cmSepaClampnCutterAxisX.commandConfiguration.fastStop.jerk := -1.0;
   cmSepaClampnCutterAxisX.commandConfiguration.fastStop.abortAcceleration := FALSE;
   cmSepaClampnCutterAxisX.commandConfiguration.fastStop.replaceStopPossible := FALSE;
   cmSepaClampnCutterAxisX.commandConfiguration.torqueLimiting.limit := -1.0;
   cmSepaClampnCutterAxisX.commandConfiguration.torqueLimiting.mode := 0;
   cmSepaClampnCutterAxisX.commandConfiguration.posRelative.distance := 0.0;
   cmSepaClampnCutterAxisX.commandConfiguration.posRelative.velocity := -1.0;
   cmSepaClampnCutterAxisX.commandConfiguration.posRelative.acceleration := -1.0;
   cmSepaClampnCutterAxisX.commandConfiguration.posRelative.deceleration := -1.0;
   cmSepaClampnCutterAxisX.commandConfiguration.posRelative.jerk := -1.0;
   cmSepaClampnCutterAxisX.commandConfiguration.posRelative.direction := 0;
   cmSepaClampnCutterAxisX.commandConfiguration.posAbsolute.position := 0.0;
   cmSepaClampnCutterAxisX.commandConfiguration.posAbsolute.velocity := -1.0;
   cmSepaClampnCutterAxisX.commandConfiguration.posAbsolute.acceleration := -1.0;
   cmSepaClampnCutterAxisX.commandConfiguration.posAbsolute.deceleration := -1.0;
   cmSepaClampnCutterAxisX.commandConfiguration.posAbsolute.jerk := -1.0;
   cmSepaClampnCutterAxisX.commandConfiguration.posAbsolute.direction := 1;
   cmSepaClampnCutterAxisX.commandConfiguration.posAbsolute.positionChangeOnTheFly := FALSE;
   cmSepaClampnCutterAxisX.commandConfiguration.posAbsolute.velocityChangeOnTheFly := FALSE;
   cmSepaClampnCutterAxisX.commandConfiguration.posSuperimposed.distance := 0.0;
   cmSepaClampnCutterAxisX.commandConfiguration.posSuperimposed.velocityDiff := -1.0;
   cmSepaClampnCutterAxisX.commandConfiguration.posSuperimposed.acceleration := -1.0;
   cmSepaClampnCutterAxisX.commandConfiguration.posSuperimposed.deceleration := -1.0;
   cmSepaClampnCutterAxisX.commandConfiguration.posSuperimposed.jerk := -1.0;
   cmSepaClampnCutterAxisX.commandConfiguration.posSuperimposed.direction := 0;
   cmSepaClampnCutterAxisX.commandConfiguration.haltSuperimposed.deceleration := -1.0;
   cmSepaClampnCutterAxisX.commandConfiguration.haltSuperimposed.jerk := -1.0;
   cmSepaClampnCutterAxisX.commandConfiguration.haltSuperimposed.abortAcceleration := FALSE;
   cmSepaClampnCutterAxisX.commandConfiguration.gearInRelative.ratioNumerator := 1;
   cmSepaClampnCutterAxisX.commandConfiguration.gearInRelative.ratioDenominator := 1;
   cmSepaClampnCutterAxisX.commandConfiguration.gearInRelative.acceleration := -1.0;
   cmSepaClampnCutterAxisX.commandConfiguration.gearInRelative.deceleration := -1.0;
   cmSepaClampnCutterAxisX.commandConfiguration.gearInRelative.jerk := -1.0;
   cmSepaClampnCutterAxisX.commandConfiguration.gearInRelative.ratioChangeOnTheFly := FALSE;
   cmSepaClampnCutterAxisX.commandConfiguration.gearInAbsolute.ratioNumerator := 1;
   cmSepaClampnCutterAxisX.commandConfiguration.gearInAbsolute.ratioDenominator := 1;
   cmSepaClampnCutterAxisX.commandConfiguration.gearInAbsolute.masterSyncPosition := 0.0;
   cmSepaClampnCutterAxisX.commandConfiguration.gearInAbsolute.slaveSyncPosition := 0.0;
   cmSepaClampnCutterAxisX.commandConfiguration.gearInAbsolute.syncProfileReference := 1;
   cmSepaClampnCutterAxisX.commandConfiguration.gearInAbsolute.masterStartDistance := 0.0;
   cmSepaClampnCutterAxisX.commandConfiguration.gearInAbsolute.velocity := -1.0;
   cmSepaClampnCutterAxisX.commandConfiguration.gearInAbsolute.acceleration := -1.0;
   cmSepaClampnCutterAxisX.commandConfiguration.gearInAbsolute.deceleration := -1.0;
   cmSepaClampnCutterAxisX.commandConfiguration.gearInAbsolute.jerk := -1.0;
   cmSepaClampnCutterAxisX.commandConfiguration.gearInAbsolute.syncDirection := 1;
   cmSepaClampnCutterAxisX.commandConfiguration.gearInAbsolute.ratioChangeOnTheFly := FALSE;
   cmSepaClampnCutterAxisX.commandConfiguration.gearInVelocity.continuousUpdate := FALSE;
   cmSepaClampnCutterAxisX.commandConfiguration.gearInVelocity.ratioNumerator := 1;
   cmSepaClampnCutterAxisX.commandConfiguration.gearInVelocity.ratioDenominator := 1;
   cmSepaClampnCutterAxisX.commandConfiguration.gearInVelocity.acceleration := -1.0;
   cmSepaClampnCutterAxisX.commandConfiguration.gearInVelocity.deceleration := -1.0;
   cmSepaClampnCutterAxisX.commandConfiguration.gearInVelocity.jerk := -1.0;
   cmSepaClampnCutterAxisX.commandConfiguration.gearInVelocity.positionControlled := FALSE;
   cmSepaClampnCutterAxisX.commandConfiguration.camIn.masterOffset := 0.0;
   cmSepaClampnCutterAxisX.commandConfiguration.camIn.slaveOffset := 0.0;
   cmSepaClampnCutterAxisX.commandConfiguration.camIn.masterScaling := 1.0;
   cmSepaClampnCutterAxisX.commandConfiguration.camIn.slaveScaling := 1.0;
   cmSepaClampnCutterAxisX.commandConfiguration.camIn.masterSyncPosition := 0.0;
   cmSepaClampnCutterAxisX.commandConfiguration.camIn.syncProfileReference := 1;
   cmSepaClampnCutterAxisX.commandConfiguration.camIn.masterStartDistance := 0.0;
   cmSepaClampnCutterAxisX.commandConfiguration.camIn.velocity := -1.0;
   cmSepaClampnCutterAxisX.commandConfiguration.camIn.acceleration := -1.0;
   cmSepaClampnCutterAxisX.commandConfiguration.camIn.deceleration := -1.0;
   cmSepaClampnCutterAxisX.commandConfiguration.camIn.jerk := -1.0;
   cmSepaClampnCutterAxisX.commandConfiguration.camIn.applicationMode := 0;
   cmSepaClampnCutterAxisX.commandConfiguration.camIn.syncDirection := 1;
   cmSepaClampnCutterAxisX.commandConfiguration.gearOutCamOut.slavePosition := 0.0;
   cmSepaClampnCutterAxisX.commandConfiguration.gearOutCamOut.syncProfileReference := 1;
   cmSepaClampnCutterAxisX.commandConfiguration.gearOutCamOut.masterStopDistance := 0.0;
   cmSepaClampnCutterAxisX.commandConfiguration.gearOutCamOut.deceleration := -1.0;
   cmSepaClampnCutterAxisX.commandConfiguration.gearOutCamOut.jerk := -1.0;
   cmSepaClampnCutterAxisX.commandConfiguration.gearOutCamOut.syncOutDirection := 3;
   cmSepaClampnCutterAxisX.commandConfiguration.gearOutCamOut.gearOutCamOutMode := -1;
   cmSepaClampnCutterAxisX.commandConfiguration.phasing.phaseShift := 0.0;
   cmSepaClampnCutterAxisX.commandConfiguration.phasing.velocity := -1.0;
   cmSepaClampnCutterAxisX.commandConfiguration.phasing.acceleration := -1.0;
   cmSepaClampnCutterAxisX.commandConfiguration.phasing.deceleration := -1.0;
   cmSepaClampnCutterAxisX.commandConfiguration.phasing.jerk := -1.0;
   cmSepaClampnCutterAxisX.commandConfiguration.phasing.profileReference := 0;
   cmSepaClampnCutterAxisX.commandConfiguration.phasing.phasingDistance := 0.0;
   cmSepaClampnCutterAxisX.commandConfiguration.phasing.startPosition := 0.0;
   cmSepaClampnCutterAxisX.commandConfiguration.phasing.direction := 3;
   cmSepaClampnCutterAxisX.commandConfiguration.phasing.phaseAbsolute := TRUE;
   cmSepaClampnCutterAxisX.commandConfiguration.phasing.phaseShiftChangeOnTheFly := FALSE;
   cmSepaClampnCutterAxisX.commandConfiguration.offset.offset := 0.0;
   cmSepaClampnCutterAxisX.commandConfiguration.offset.profileReference := 1;
   cmSepaClampnCutterAxisX.commandConfiguration.offset.offsetDistance := 0.0;
   cmSepaClampnCutterAxisX.commandConfiguration.offset.startPosition := 0.0;
   cmSepaClampnCutterAxisX.commandConfiguration.offset.direction := 3;
   cmSepaClampnCutterAxisX.commandConfiguration.offset.offsetAbsolute := TRUE;
   cmSepaClampnCutterAxisX.commandConfiguration.offset.offsetChangeOnTheFly := FALSE;
   cmSepaClampnCutterAxisZ.commandConfiguration.generalSettings.stopOnError := TRUE;
   cmSepaClampnCutterAxisZ.commandConfiguration.generalSettings.resetWithRestart := FALSE;
   cmSepaClampnCutterAxisZ.commandConfiguration.generalSettings.abortWaitingSyncCmd := TRUE;
   cmSepaClampnCutterAxisZ.commandConfiguration.power.startMode := 1;
   cmSepaClampnCutterAxisZ.commandConfiguration.power.stopMode := 0;
   cmSepaClampnCutterAxisZ.commandConfiguration.power.syncMotionSimulation := FALSE;
   cmSepaClampnCutterAxisZ.commandConfiguration.power.syncMotionSimulationExtendedMode := -1;
   cmSepaClampnCutterAxisZ.commandConfiguration.jog.velocity := 0.0;
   cmSepaClampnCutterAxisZ.commandConfiguration.jog.acceleration := -1.0;
   cmSepaClampnCutterAxisZ.commandConfiguration.jog.deceleration := -1.0;
   cmSepaClampnCutterAxisZ.commandConfiguration.jog.jerk := -1.0;
   cmSepaClampnCutterAxisZ.commandConfiguration.jog.positionControlled := TRUE;
   cmSepaClampnCutterAxisZ.commandConfiguration.jog.increment := 0.0;
   cmSepaClampnCutterAxisZ.commandConfiguration.jog.mode := 0;
   cmSepaClampnCutterAxisZ.commandConfiguration.moveVelocity.velocity := 0.0;
   cmSepaClampnCutterAxisZ.commandConfiguration.moveVelocity.acceleration := -1.0;
   cmSepaClampnCutterAxisZ.commandConfiguration.moveVelocity.deceleration := -1.0;
   cmSepaClampnCutterAxisZ.commandConfiguration.moveVelocity.jerk := -1.0;
   cmSepaClampnCutterAxisZ.commandConfiguration.moveVelocity.direction := 0;
   cmSepaClampnCutterAxisZ.commandConfiguration.moveVelocity.positionControlled := TRUE;
   cmSepaClampnCutterAxisZ.commandConfiguration.moveVelocity.velocityChangeOnTheFly := FALSE;
   cmSepaClampnCutterAxisZ.commandConfiguration.stop.deceleration := -1.0;
   cmSepaClampnCutterAxisZ.commandConfiguration.stop.jerk := -1.0;
   cmSepaClampnCutterAxisZ.commandConfiguration.stop.abortAcceleration := FALSE;
   cmSepaClampnCutterAxisZ.commandConfiguration.fastStop.deceleration := -1.0;
   cmSepaClampnCutterAxisZ.commandConfiguration.fastStop.jerk := -1.0;
   cmSepaClampnCutterAxisZ.commandConfiguration.fastStop.abortAcceleration := FALSE;
   cmSepaClampnCutterAxisZ.commandConfiguration.fastStop.replaceStopPossible := FALSE;
   cmSepaClampnCutterAxisZ.commandConfiguration.torqueLimiting.limit := -1.0;
   cmSepaClampnCutterAxisZ.commandConfiguration.torqueLimiting.mode := 0;
   cmSepaClampnCutterAxisZ.commandConfiguration.homing.position := 0.0;
   cmSepaClampnCutterAxisZ.commandConfiguration.homing.mode := 0;
   cmSepaClampnCutterAxisZ.commandConfiguration.homing.sensor := 0;
   cmSepaClampnCutterAxisZ.commandConfiguration.homing.extendedMode := -1;
   cmSepaClampnCutterAxisZ.commandConfiguration.homing.extendedModeTorqueLimit := 0.0;
   cmSepaClampnCutterAxisZ.commandConfiguration.homing.extendedModeTargetPosition := 0.0;
   cmSepaClampnCutterAxisZ.commandConfiguration.posRelative.distance := 0.0;
   cmSepaClampnCutterAxisZ.commandConfiguration.posRelative.velocity := -1.0;
   cmSepaClampnCutterAxisZ.commandConfiguration.posRelative.acceleration := -1.0;
   cmSepaClampnCutterAxisZ.commandConfiguration.posRelative.deceleration := -1.0;
   cmSepaClampnCutterAxisZ.commandConfiguration.posRelative.jerk := -1.0;
   cmSepaClampnCutterAxisZ.commandConfiguration.posRelative.direction := 0;
   cmSepaClampnCutterAxisZ.commandConfiguration.posAbsolute.position := 0.0;
   cmSepaClampnCutterAxisZ.commandConfiguration.posAbsolute.velocity := -1.0;
   cmSepaClampnCutterAxisZ.commandConfiguration.posAbsolute.acceleration := -1.0;
   cmSepaClampnCutterAxisZ.commandConfiguration.posAbsolute.deceleration := -1.0;
   cmSepaClampnCutterAxisZ.commandConfiguration.posAbsolute.jerk := -1.0;
   cmSepaClampnCutterAxisZ.commandConfiguration.posAbsolute.direction := 1;
   cmSepaClampnCutterAxisZ.commandConfiguration.posAbsolute.positionChangeOnTheFly := FALSE;
   cmSepaClampnCutterAxisZ.commandConfiguration.posAbsolute.velocityChangeOnTheFly := FALSE;
   cmSepaClampnCutterAxisZ.commandConfiguration.posSuperimposed.distance := 0.0;
   cmSepaClampnCutterAxisZ.commandConfiguration.posSuperimposed.velocityDiff := -1.0;
   cmSepaClampnCutterAxisZ.commandConfiguration.posSuperimposed.acceleration := -1.0;
   cmSepaClampnCutterAxisZ.commandConfiguration.posSuperimposed.deceleration := -1.0;
   cmSepaClampnCutterAxisZ.commandConfiguration.posSuperimposed.jerk := -1.0;
   cmSepaClampnCutterAxisZ.commandConfiguration.posSuperimposed.direction := 0;
   cmSepaClampnCutterAxisZ.commandConfiguration.haltSuperimposed.deceleration := -1.0;
   cmSepaClampnCutterAxisZ.commandConfiguration.haltSuperimposed.jerk := -1.0;
   cmSepaClampnCutterAxisZ.commandConfiguration.haltSuperimposed.abortAcceleration := FALSE;
   cmSepaClampnCutterAxisZ.commandConfiguration.gearInRelative.ratioNumerator := 1;
   cmSepaClampnCutterAxisZ.commandConfiguration.gearInRelative.ratioDenominator := 1;
   cmSepaClampnCutterAxisZ.commandConfiguration.gearInRelative.acceleration := -1.0;
   cmSepaClampnCutterAxisZ.commandConfiguration.gearInRelative.deceleration := -1.0;
   cmSepaClampnCutterAxisZ.commandConfiguration.gearInRelative.jerk := -1.0;
   cmSepaClampnCutterAxisZ.commandConfiguration.gearInRelative.ratioChangeOnTheFly := FALSE;
   cmSepaClampnCutterAxisZ.commandConfiguration.gearInAbsolute.ratioNumerator := 1;
   cmSepaClampnCutterAxisZ.commandConfiguration.gearInAbsolute.ratioDenominator := 1;
   cmSepaClampnCutterAxisZ.commandConfiguration.gearInAbsolute.masterSyncPosition := 0.0;
   cmSepaClampnCutterAxisZ.commandConfiguration.gearInAbsolute.slaveSyncPosition := 0.0;
   cmSepaClampnCutterAxisZ.commandConfiguration.gearInAbsolute.syncProfileReference := 1;
   cmSepaClampnCutterAxisZ.commandConfiguration.gearInAbsolute.masterStartDistance := 0.0;
   cmSepaClampnCutterAxisZ.commandConfiguration.gearInAbsolute.velocity := -1.0;
   cmSepaClampnCutterAxisZ.commandConfiguration.gearInAbsolute.acceleration := -1.0;
   cmSepaClampnCutterAxisZ.commandConfiguration.gearInAbsolute.deceleration := -1.0;
   cmSepaClampnCutterAxisZ.commandConfiguration.gearInAbsolute.jerk := -1.0;
   cmSepaClampnCutterAxisZ.commandConfiguration.gearInAbsolute.syncDirection := 1;
   cmSepaClampnCutterAxisZ.commandConfiguration.gearInAbsolute.ratioChangeOnTheFly := FALSE;
   cmSepaClampnCutterAxisZ.commandConfiguration.gearInVelocity.continuousUpdate := FALSE;
   cmSepaClampnCutterAxisZ.commandConfiguration.gearInVelocity.ratioNumerator := 1;
   cmSepaClampnCutterAxisZ.commandConfiguration.gearInVelocity.ratioDenominator := 1;
   cmSepaClampnCutterAxisZ.commandConfiguration.gearInVelocity.acceleration := -1.0;
   cmSepaClampnCutterAxisZ.commandConfiguration.gearInVelocity.deceleration := -1.0;
   cmSepaClampnCutterAxisZ.commandConfiguration.gearInVelocity.jerk := -1.0;
   cmSepaClampnCutterAxisZ.commandConfiguration.gearInVelocity.positionControlled := FALSE;
   cmSepaClampnCutterAxisZ.commandConfiguration.camIn.masterOffset := 0.0;
   cmSepaClampnCutterAxisZ.commandConfiguration.camIn.slaveOffset := 0.0;
   cmSepaClampnCutterAxisZ.commandConfiguration.camIn.masterScaling := 1.0;
   cmSepaClampnCutterAxisZ.commandConfiguration.camIn.slaveScaling := 1.0;
   cmSepaClampnCutterAxisZ.commandConfiguration.camIn.masterSyncPosition := 0.0;
   cmSepaClampnCutterAxisZ.commandConfiguration.camIn.syncProfileReference := 1;
   cmSepaClampnCutterAxisZ.commandConfiguration.camIn.masterStartDistance := 0.0;
   cmSepaClampnCutterAxisZ.commandConfiguration.camIn.velocity := -1.0;
   cmSepaClampnCutterAxisZ.commandConfiguration.camIn.acceleration := -1.0;
   cmSepaClampnCutterAxisZ.commandConfiguration.camIn.deceleration := -1.0;
   cmSepaClampnCutterAxisZ.commandConfiguration.camIn.jerk := -1.0;
   cmSepaClampnCutterAxisZ.commandConfiguration.camIn.applicationMode := 0;
   cmSepaClampnCutterAxisZ.commandConfiguration.camIn.syncDirection := 1;
   cmSepaClampnCutterAxisZ.commandConfiguration.gearOutCamOut.slavePosition := 0.0;
   cmSepaClampnCutterAxisZ.commandConfiguration.gearOutCamOut.syncProfileReference := 1;
   cmSepaClampnCutterAxisZ.commandConfiguration.gearOutCamOut.masterStopDistance := 0.0;
   cmSepaClampnCutterAxisZ.commandConfiguration.gearOutCamOut.deceleration := -1.0;
   cmSepaClampnCutterAxisZ.commandConfiguration.gearOutCamOut.jerk := -1.0;
   cmSepaClampnCutterAxisZ.commandConfiguration.gearOutCamOut.syncOutDirection := 3;
   cmSepaClampnCutterAxisZ.commandConfiguration.gearOutCamOut.gearOutCamOutMode := -1;
   cmSepaClampnCutterAxisZ.commandConfiguration.phasing.phaseShift := 0.0;
   cmSepaClampnCutterAxisZ.commandConfiguration.phasing.velocity := -1.0;
   cmSepaClampnCutterAxisZ.commandConfiguration.phasing.acceleration := -1.0;
   cmSepaClampnCutterAxisZ.commandConfiguration.phasing.deceleration := -1.0;
   cmSepaClampnCutterAxisZ.commandConfiguration.phasing.jerk := -1.0;
   cmSepaClampnCutterAxisZ.commandConfiguration.phasing.profileReference := 0;
   cmSepaClampnCutterAxisZ.commandConfiguration.phasing.phasingDistance := 0.0;
   cmSepaClampnCutterAxisZ.commandConfiguration.phasing.startPosition := 0.0;
   cmSepaClampnCutterAxisZ.commandConfiguration.phasing.direction := 3;
   cmSepaClampnCutterAxisZ.commandConfiguration.phasing.phaseAbsolute := TRUE;
   cmSepaClampnCutterAxisZ.commandConfiguration.phasing.phaseShiftChangeOnTheFly := FALSE;
   cmSepaClampnCutterAxisZ.commandConfiguration.offset.offset := 0.0;
   cmSepaClampnCutterAxisZ.commandConfiguration.offset.profileReference := 1;
   cmSepaClampnCutterAxisZ.commandConfiguration.offset.offsetDistance := 0.0;
   cmSepaClampnCutterAxisZ.commandConfiguration.offset.startPosition := 0.0;
   cmSepaClampnCutterAxisZ.commandConfiguration.offset.direction := 3;
   cmSepaClampnCutterAxisZ.commandConfiguration.offset.offsetAbsolute := TRUE;
   cmSepaClampnCutterAxisZ.commandConfiguration.offset.offsetChangeOnTheFly := FALSE;
   cmSepaClampnCutterAxisZ.commands.enableAxis := FALSE;
   cmSepaClampnCutterAxisZ.commands.resetAxis := FALSE;
   cmSepaClampnCutterAxisZ.commands.openBrake := FALSE;
   cmSepaClampnCutterAxisZ.commands.jogForward := FALSE;
   cmSepaClampnCutterAxisZ.commands.jogBackward := FALSE;
   cmSepaClampnCutterAxisZ.commands.moveVelocity := FALSE;
   cmSepaClampnCutterAxisZ.commands.stop := FALSE;
   cmSepaClampnCutterAxisZ.commands.fastStop := FALSE;
   cmSepaClampnCutterAxisZ.commands.torqueLimiting := FALSE;
   cmSepaClampnCutterAxisZ.commands.homing := FALSE;
   cmSepaClampnCutterAxisZ.commands.posRelative := FALSE;
   cmSepaClampnCutterAxisZ.commands.posAbsolute := FALSE;
   cmSepaClampnCutterAxisZ.commands.posSuperimposed := FALSE;
   cmSepaClampnCutterAxisZ.commands.haltSuperimposed := FALSE;
   cmSepaClampnCutterAxisZ.commands.selectSetPosition := -1;
   cmSepaClampnCutterAxisZ.commands.reset := FALSE;
   cmSepaGripperAxisX.commandConfiguration.stop.deceleration := -1.0;
   cmSepaGripperAxisX.commandConfiguration.stop.jerk := -1.0;
   cmSepaGripperAxisX.commandConfiguration.stop.abortAcceleration := FALSE;
   cmSepaGripperAxisX.commandConfiguration.fastStop.deceleration := -1.0;
   cmSepaGripperAxisX.commandConfiguration.fastStop.jerk := -1.0;
   cmSepaGripperAxisX.commandConfiguration.fastStop.abortAcceleration := FALSE;
   cmSepaGripperAxisX.commandConfiguration.fastStop.replaceStopPossible := FALSE;
   cmSepaGripperAxisX.commandConfiguration.torqueLimiting.limit := -1.0;
   cmSepaGripperAxisX.commandConfiguration.torqueLimiting.mode := 0;
   cmSepaGripperAxisX.commandConfiguration.homing.position := 0.0;
   cmSepaGripperAxisX.commandConfiguration.homing.mode := 0;
   cmSepaGripperAxisX.commandConfiguration.homing.sensor := 0;
   cmSepaGripperAxisX.commandConfiguration.homing.extendedMode := -1;
   cmSepaGripperAxisX.commandConfiguration.homing.extendedModeTorqueLimit := 0.0;
   cmSepaGripperAxisX.commandConfiguration.homing.extendedModeTargetPosition := 0.0;
   cmSepaGripperAxisX.commandConfiguration.posRelative.distance := 0.0;
   cmSepaGripperAxisX.commandConfiguration.posRelative.velocity := -1.0;
   cmSepaGripperAxisX.commandConfiguration.posRelative.acceleration := -1.0;
   cmSepaGripperAxisX.commandConfiguration.posRelative.deceleration := -1.0;
   cmSepaGripperAxisX.commandConfiguration.posRelative.jerk := -1.0;
   cmSepaGripperAxisX.commandConfiguration.posRelative.direction := 0;
   cmSepaGripperAxisX.commandConfiguration.posAbsolute.position := 0.0;
   cmSepaGripperAxisX.commandConfiguration.posAbsolute.velocity := -1.0;
   cmSepaGripperAxisX.commandConfiguration.posAbsolute.acceleration := -1.0;
   cmSepaGripperAxisX.commandConfiguration.posAbsolute.deceleration := -1.0;
   cmSepaGripperAxisX.commandConfiguration.posAbsolute.jerk := -1.0;
   cmSepaGripperAxisX.commandConfiguration.posAbsolute.direction := 1;
   cmSepaGripperAxisX.commandConfiguration.posAbsolute.positionChangeOnTheFly := FALSE;
   cmSepaGripperAxisX.commandConfiguration.posAbsolute.velocityChangeOnTheFly := FALSE;
   cmSepaGripperAxisX.commandConfiguration.posSuperimposed.distance := 0.0;
   cmSepaGripperAxisX.commandConfiguration.posSuperimposed.velocityDiff := -1.0;
   cmSepaGripperAxisX.commandConfiguration.posSuperimposed.acceleration := -1.0;
   cmSepaGripperAxisX.commandConfiguration.posSuperimposed.deceleration := -1.0;
   cmSepaGripperAxisX.commandConfiguration.posSuperimposed.jerk := -1.0;
   cmSepaGripperAxisX.commandConfiguration.posSuperimposed.direction := 0;
   cmSepaGripperAxisX.commandConfiguration.haltSuperimposed.deceleration := -1.0;
   cmSepaGripperAxisX.commandConfiguration.haltSuperimposed.jerk := -1.0;
   cmSepaGripperAxisX.commandConfiguration.haltSuperimposed.abortAcceleration := FALSE;
   cmSepaGripperAxisX.commandConfiguration.gearInRelative.ratioNumerator := 1;
   cmSepaGripperAxisX.commandConfiguration.gearInRelative.ratioDenominator := 1;
   cmSepaGripperAxisX.commandConfiguration.gearInRelative.acceleration := -1.0;
   cmSepaGripperAxisX.commandConfiguration.gearInRelative.deceleration := -1.0;
   cmSepaGripperAxisX.commandConfiguration.gearInRelative.jerk := -1.0;
   cmSepaGripperAxisX.commandConfiguration.gearInRelative.ratioChangeOnTheFly := FALSE;
   cmSepaGripperAxisX.commandConfiguration.gearInAbsolute.ratioNumerator := 1;
   cmSepaGripperAxisX.commandConfiguration.gearInAbsolute.ratioDenominator := 1;
   cmSepaGripperAxisX.commandConfiguration.gearInAbsolute.masterSyncPosition := 0.0;
   cmSepaGripperAxisX.commandConfiguration.gearInAbsolute.slaveSyncPosition := 0.0;
   cmSepaGripperAxisX.commandConfiguration.gearInAbsolute.syncProfileReference := 1;
   cmSepaGripperAxisX.commandConfiguration.gearInAbsolute.masterStartDistance := 0.0;
   cmSepaGripperAxisX.commandConfiguration.gearInAbsolute.velocity := -1.0;
   cmSepaGripperAxisX.commandConfiguration.gearInAbsolute.acceleration := -1.0;
   cmSepaGripperAxisX.commandConfiguration.gearInAbsolute.deceleration := -1.0;
   cmSepaGripperAxisX.commandConfiguration.gearInAbsolute.jerk := -1.0;
   cmSepaGripperAxisX.commandConfiguration.gearInAbsolute.syncDirection := 1;
   cmSepaGripperAxisX.commandConfiguration.gearInAbsolute.ratioChangeOnTheFly := FALSE;
   cmSepaGripperAxisX.commandConfiguration.gearInVelocity.continuousUpdate := FALSE;
   cmSepaGripperAxisX.commandConfiguration.gearInVelocity.ratioNumerator := 1;
   cmSepaGripperAxisX.commandConfiguration.gearInVelocity.ratioDenominator := 1;
   cmSepaGripperAxisX.commandConfiguration.gearInVelocity.acceleration := -1.0;
   cmSepaGripperAxisX.commandConfiguration.gearInVelocity.deceleration := -1.0;
   cmSepaGripperAxisX.commandConfiguration.gearInVelocity.jerk := -1.0;
   cmSepaGripperAxisX.commandConfiguration.gearInVelocity.positionControlled := FALSE;
   cmSepaGripperAxisX.commandConfiguration.camIn.masterOffset := 0.0;
   cmSepaGripperAxisX.commandConfiguration.camIn.slaveOffset := 0.0;
   cmSepaGripperAxisX.commandConfiguration.camIn.masterScaling := 1.0;
   cmSepaGripperAxisX.commandConfiguration.camIn.slaveScaling := 1.0;
   cmSepaGripperAxisX.commandConfiguration.camIn.masterSyncPosition := 0.0;
   cmSepaGripperAxisX.commandConfiguration.camIn.syncProfileReference := 1;
   cmSepaGripperAxisX.commandConfiguration.camIn.masterStartDistance := 0.0;
   cmSepaGripperAxisX.commandConfiguration.camIn.velocity := -1.0;
   cmSepaGripperAxisX.commandConfiguration.camIn.acceleration := -1.0;
   cmSepaGripperAxisX.commandConfiguration.camIn.deceleration := -1.0;
   cmSepaGripperAxisX.commandConfiguration.camIn.jerk := -1.0;
   cmSepaGripperAxisX.commandConfiguration.camIn.applicationMode := 0;
   cmSepaGripperAxisX.commandConfiguration.camIn.syncDirection := 1;
   cmSepaGripperAxisX.commandConfiguration.gearOutCamOut.slavePosition := 0.0;
   cmSepaGripperAxisX.commandConfiguration.gearOutCamOut.syncProfileReference := 1;
   cmSepaGripperAxisX.commandConfiguration.gearOutCamOut.masterStopDistance := 0.0;
   cmSepaGripperAxisX.commandConfiguration.gearOutCamOut.deceleration := -1.0;
   cmSepaGripperAxisX.commandConfiguration.gearOutCamOut.jerk := -1.0;
   cmSepaGripperAxisX.commandConfiguration.gearOutCamOut.syncOutDirection := 3;
   cmSepaGripperAxisX.commandConfiguration.gearOutCamOut.gearOutCamOutMode := -1;
   cmSepaGripperAxisX.commandConfiguration.phasing.phaseShift := 0.0;
   cmSepaGripperAxisX.commandConfiguration.phasing.velocity := -1.0;
   cmSepaGripperAxisX.commandConfiguration.phasing.acceleration := -1.0;
   cmSepaGripperAxisX.commandConfiguration.phasing.deceleration := -1.0;
   cmSepaGripperAxisX.commandConfiguration.phasing.jerk := -1.0;
   cmSepaGripperAxisX.commandConfiguration.phasing.profileReference := 0;
   cmSepaGripperAxisX.commandConfiguration.phasing.phasingDistance := 0.0;
   cmSepaGripperAxisX.commandConfiguration.phasing.startPosition := 0.0;
   cmSepaGripperAxisX.commandConfiguration.phasing.direction := 3;
   cmSepaGripperAxisX.commandConfiguration.phasing.phaseAbsolute := TRUE;
   cmSepaGripperAxisX.commandConfiguration.phasing.phaseShiftChangeOnTheFly := FALSE;
   cmSepaGripperAxisX.commandConfiguration.offset.offset := 0.0;
   cmSepaGripperAxisX.commandConfiguration.offset.profileReference := 1;
   cmSepaGripperAxisX.commandConfiguration.offset.offsetDistance := 0.0;
   cmSepaGripperAxisX.commandConfiguration.offset.startPosition := 0.0;
   cmSepaGripperAxisX.commandConfiguration.offset.direction := 3;
   cmSepaGripperAxisX.commandConfiguration.offset.offsetAbsolute := TRUE;
   cmSepaGripperAxisX.commandConfiguration.offset.offsetChangeOnTheFly := FALSE;
   cmSepaGripperAxisZ.commandConfiguration.generalSettings.stopOnError := TRUE;
   cmSepaGripperAxisZ.commandConfiguration.generalSettings.resetWithRestart := FALSE;
   cmSepaGripperAxisZ.commandConfiguration.generalSettings.abortWaitingSyncCmd := TRUE;
   cmSepaGripperAxisZ.commandConfiguration.power.startMode := 1;
   cmSepaGripperAxisZ.commandConfiguration.power.stopMode := 0;
   cmSepaGripperAxisZ.commandConfiguration.power.syncMotionSimulation := FALSE;
   cmSepaGripperAxisZ.commandConfiguration.power.syncMotionSimulationExtendedMode := -1;
   cmSepaGripperAxisZ.commandConfiguration.jog.velocity := 0.0;
   cmSepaGripperAxisZ.commandConfiguration.jog.acceleration := -1.0;
   cmSepaGripperAxisZ.commandConfiguration.jog.deceleration := -1.0;
   cmSepaGripperAxisZ.commandConfiguration.jog.jerk := -1.0;
   cmSepaGripperAxisZ.commandConfiguration.jog.positionControlled := TRUE;
   cmSepaGripperAxisZ.commandConfiguration.jog.increment := 0.0;
   cmSepaGripperAxisZ.commandConfiguration.jog.mode := 0;
   cmSepaGripperAxisZ.commandConfiguration.moveVelocity.velocity := 0.0;
   cmSepaGripperAxisZ.commandConfiguration.moveVelocity.acceleration := -1.0;
   cmSepaGripperAxisZ.commandConfiguration.moveVelocity.deceleration := -1.0;
   cmSepaGripperAxisZ.commandConfiguration.moveVelocity.jerk := -1.0;
   cmSepaGripperAxisZ.commandConfiguration.moveVelocity.direction := 0;
   cmSepaGripperAxisZ.commandConfiguration.moveVelocity.positionControlled := TRUE;
   cmSepaGripperAxisZ.commandConfiguration.moveVelocity.velocityChangeOnTheFly := FALSE;
   cmSepaGripperAxisZ.commandConfiguration.stop.deceleration := -1.0;
   cmSepaGripperAxisZ.commandConfiguration.stop.jerk := -1.0;
   cmSepaGripperAxisZ.commandConfiguration.stop.abortAcceleration := FALSE;
   cmSepaGripperAxisZ.commandConfiguration.fastStop.deceleration := -1.0;
   cmSepaGripperAxisZ.commandConfiguration.fastStop.jerk := -1.0;
   cmSepaGripperAxisZ.commandConfiguration.fastStop.abortAcceleration := FALSE;
   cmSepaGripperAxisZ.commandConfiguration.fastStop.replaceStopPossible := FALSE;
   cmSepaGripperAxisZ.commandConfiguration.torqueLimiting.limit := -1.0;
   cmSepaGripperAxisZ.commandConfiguration.torqueLimiting.mode := 0;
   cmSepaGripperAxisZ.commandConfiguration.homing.position := 0.0;
   cmSepaGripperAxisZ.commandConfiguration.homing.mode := 0;
   cmSepaGripperAxisZ.commandConfiguration.homing.sensor := 0;
   cmSepaGripperAxisZ.commandConfiguration.homing.extendedMode := -1;
   cmSepaGripperAxisZ.commandConfiguration.homing.extendedModeTorqueLimit := 0.0;
   cmSepaGripperAxisZ.commandConfiguration.homing.extendedModeTargetPosition := 0.0;
   cmSepaGripperAxisZ.commandConfiguration.posRelative.distance := 0.0;
   cmSepaGripperAxisZ.commandConfiguration.posRelative.velocity := -1.0;
   cmSepaGripperAxisZ.commandConfiguration.posRelative.acceleration := -1.0;
   cmSepaGripperAxisZ.commandConfiguration.posRelative.deceleration := -1.0;
   cmSepaGripperAxisZ.commandConfiguration.posRelative.jerk := -1.0;
   cmSepaGripperAxisZ.commandConfiguration.posRelative.direction := 0;
   cmSepaGripperAxisZ.commandConfiguration.posAbsolute.position := 0.0;
   cmSepaGripperAxisZ.commandConfiguration.posAbsolute.velocity := -1.0;
   cmSepaGripperAxisZ.commandConfiguration.posAbsolute.acceleration := -1.0;
   cmSepaGripperAxisZ.commandConfiguration.posAbsolute.deceleration := -1.0;
   cmSepaGripperAxisZ.commandConfiguration.posAbsolute.jerk := -1.0;
   cmSepaGripperAxisZ.commandConfiguration.posAbsolute.direction := 1;
   cmSepaGripperAxisZ.commandConfiguration.posAbsolute.positionChangeOnTheFly := FALSE;
   cmSepaGripperAxisZ.commandConfiguration.posAbsolute.velocityChangeOnTheFly := FALSE;
   cmSepaGripperAxisZ.commandConfiguration.posSuperimposed.distance := 0.0;
   cmSepaGripperAxisZ.commandConfiguration.posSuperimposed.velocityDiff := -1.0;
   cmSepaGripperAxisZ.commandConfiguration.posSuperimposed.acceleration := -1.0;
   cmSepaGripperAxisZ.commandConfiguration.posSuperimposed.deceleration := -1.0;
   cmSepaGripperAxisZ.commandConfiguration.posSuperimposed.jerk := -1.0;
   cmSepaGripperAxisZ.commandConfiguration.posSuperimposed.direction := 0;
   cmSepaGripperAxisZ.commandConfiguration.haltSuperimposed.deceleration := -1.0;
   cmSepaGripperAxisZ.commandConfiguration.haltSuperimposed.jerk := -1.0;
   cmSepaGripperAxisZ.commandConfiguration.haltSuperimposed.abortAcceleration := FALSE;
   cmSepaGripperAxisZ.commandConfiguration.gearInRelative.ratioNumerator := 1;
   cmSepaGripperAxisZ.commandConfiguration.gearInRelative.ratioDenominator := 1;
   cmSepaGripperAxisZ.commandConfiguration.gearInRelative.acceleration := -1.0;
   cmSepaGripperAxisZ.commandConfiguration.gearInRelative.deceleration := -1.0;
   cmSepaGripperAxisZ.commandConfiguration.gearInRelative.jerk := -1.0;
   cmSepaGripperAxisZ.commandConfiguration.gearInRelative.ratioChangeOnTheFly := FALSE;
   cmSepaGripperAxisZ.commandConfiguration.gearInAbsolute.ratioNumerator := 1;
   cmSepaGripperAxisZ.commandConfiguration.gearInAbsolute.ratioDenominator := 1;
   cmSepaGripperAxisZ.commandConfiguration.gearInAbsolute.masterSyncPosition := 0.0;
   cmSepaGripperAxisZ.commandConfiguration.gearInAbsolute.slaveSyncPosition := 0.0;
   cmSepaGripperAxisZ.commandConfiguration.gearInAbsolute.syncProfileReference := 1;
   cmSepaGripperAxisZ.commandConfiguration.gearInAbsolute.masterStartDistance := 0.0;
   cmSepaGripperAxisZ.commandConfiguration.gearInAbsolute.velocity := -1.0;
   cmSepaGripperAxisZ.commandConfiguration.gearInAbsolute.acceleration := -1.0;
   cmSepaGripperAxisZ.commandConfiguration.gearInAbsolute.deceleration := -1.0;
   cmSepaGripperAxisZ.commandConfiguration.gearInAbsolute.jerk := -1.0;
   cmSepaGripperAxisZ.commandConfiguration.gearInAbsolute.syncDirection := 1;
   cmSepaGripperAxisZ.commandConfiguration.gearInAbsolute.ratioChangeOnTheFly := FALSE;
   cmSepaGripperAxisZ.commandConfiguration.gearInVelocity.continuousUpdate := FALSE;
   cmSepaGripperAxisZ.commandConfiguration.gearInVelocity.ratioNumerator := 1;
   cmSepaGripperAxisZ.commandConfiguration.gearInVelocity.ratioDenominator := 1;
   cmSepaGripperAxisZ.commandConfiguration.gearInVelocity.acceleration := -1.0;
   cmSepaGripperAxisZ.commandConfiguration.gearInVelocity.deceleration := -1.0;
   cmSepaGripperAxisZ.commandConfiguration.gearInVelocity.jerk := -1.0;
   cmSepaGripperAxisZ.commandConfiguration.gearInVelocity.positionControlled := FALSE;
   cmSepaGripperAxisZ.commandConfiguration.camIn.masterOffset := 0.0;
   cmSepaGripperAxisZ.commandConfiguration.camIn.slaveOffset := 0.0;
   cmSepaGripperAxisZ.commandConfiguration.camIn.masterScaling := 1.0;
   cmSepaGripperAxisZ.commandConfiguration.camIn.slaveScaling := 1.0;
   cmSepaGripperAxisZ.commandConfiguration.camIn.masterSyncPosition := 0.0;
   cmSepaGripperAxisZ.commandConfiguration.camIn.syncProfileReference := 1;
   cmSepaGripperAxisZ.commandConfiguration.camIn.masterStartDistance := 0.0;
   cmSepaGripperAxisZ.commandConfiguration.camIn.velocity := -1.0;
   cmSepaGripperAxisZ.commandConfiguration.camIn.acceleration := -1.0;
   cmSepaGripperAxisZ.commandConfiguration.camIn.deceleration := -1.0;
   cmSepaGripperAxisZ.commandConfiguration.camIn.jerk := -1.0;
   cmSepaGripperAxisZ.commandConfiguration.camIn.applicationMode := 0;
   cmSepaGripperAxisZ.commandConfiguration.camIn.syncDirection := 1;
   cmSepaGripperAxisZ.commandConfiguration.gearOutCamOut.slavePosition := 0.0;
   cmSepaGripperAxisZ.commandConfiguration.gearOutCamOut.syncProfileReference := 1;
   cmSepaGripperAxisZ.commandConfiguration.gearOutCamOut.masterStopDistance := 0.0;
   cmSepaGripperAxisZ.commandConfiguration.gearOutCamOut.deceleration := -1.0;
   cmSepaGripperAxisZ.commandConfiguration.gearOutCamOut.jerk := -1.0;
   cmSepaGripperAxisZ.commandConfiguration.gearOutCamOut.syncOutDirection := 3;
   cmSepaGripperAxisZ.commandConfiguration.gearOutCamOut.gearOutCamOutMode := -1;
   cmSepaGripperAxisZ.commandConfiguration.phasing.phaseShift := 0.0;
   cmSepaGripperAxisZ.commandConfiguration.phasing.velocity := -1.0;
   cmSepaGripperAxisZ.commandConfiguration.phasing.acceleration := -1.0;
   cmSepaGripperAxisZ.commandConfiguration.phasing.deceleration := -1.0;
   cmSepaGripperAxisZ.commandConfiguration.phasing.jerk := -1.0;
   cmSepaGripperAxisZ.commandConfiguration.phasing.profileReference := 0;
   cmSepaGripperAxisZ.commandConfiguration.phasing.phasingDistance := 0.0;
   cmSepaGripperAxisZ.commandConfiguration.phasing.startPosition := 0.0;
   cmSepaGripperAxisZ.commandConfiguration.phasing.direction := 3;
   cmSepaGripperAxisZ.commandConfiguration.phasing.phaseAbsolute := TRUE;
   cmSepaGripperAxisZ.commandConfiguration.phasing.phaseShiftChangeOnTheFly := FALSE;
   cmSepaGripperAxisZ.commandConfiguration.offset.offset := 0.0;
   cmSepaGripperAxisZ.commandConfiguration.offset.profileReference := 1;
   cmSepaGripperAxisZ.commandConfiguration.offset.offsetDistance := 0.0;
   cmSepaGripperAxisZ.commandConfiguration.offset.startPosition := 0.0;
   cmSepaGripperAxisZ.commandConfiguration.offset.direction := 3;
   cmSepaGripperAxisZ.commandConfiguration.offset.offsetAbsolute := TRUE;
   cmSepaGripperAxisZ.commandConfiguration.offset.offsetChangeOnTheFly := FALSE;
   cmSepaGripperAxisZ.commands.enableAxis := FALSE;
   cmSepaGripperAxisZ.commands.resetAxis := FALSE;
   cmSepaGripperAxisZ.commands.openBrake := FALSE;
   cmSepaGripperAxisZ.commands.jogForward := FALSE;
   cmSepaGripperAxisZ.commands.jogBackward := FALSE;
   cmSepaGripperAxisZ.commands.moveVelocity := FALSE;
   cmSepaGripperAxisZ.commands.stop := FALSE;
   cmSepaGripperAxisZ.commands.fastStop := FALSE;
   cmSepaGripperAxisZ.commands.torqueLimiting := FALSE;
   cmSepaGripperAxisZ.commands.homing := FALSE;
   cmSepaGripperAxisZ.commands.posRelative := FALSE;
   cmSepaGripperAxisZ.commands.posAbsolute := FALSE;
   cmSepaGripperAxisZ.commands.posSuperimposed := FALSE;
   cmSepaGripperAxisZ.commands.haltSuperimposed := FALSE;
   cmSepaGripperAxisZ.commands.selectSetPosition := -1;
   cmSepaGripperAxisZ.commands.reset := FALSE;
   cmSepaGripperAxisZ.monitoring.valid := FALSE;
   cmSepaGripperAxisZ.monitoring.busy := TRUE;
   cmSepaGripperAxisZ.monitoring.error := TRUE;
   cmSepaGripperAxisZ.monitoring.status := 16#8600;
   cmSepaGripperAxisZ.monitoring.subfunctionStatus := 16#8001;
   cmSepaGripperAxisZ.monitoring.axisEnabled := FALSE;
   cmSepaGripperAxisZ.monitoring.resetActive := FALSE;
   cmSepaGripperAxisZ.monitoring.inVelocity := FALSE;
   cmSepaGripperAxisZ.monitoring.inLimitation := FALSE;
   cmSepaGripperAxisZ.monitoring.inClamping := FALSE;
   cmSepaGripperAxisZ.monitoring.startSync := FALSE;
   cmSepaGripperAxisZ.monitoring.inSync := FALSE;
   cmSepaGripperAxisZ.monitoring.inSimulation := FALSE;
   cmSepaGripperAxisZ.monitoring.jogSelected := FALSE;
   cmSepaGripperAxisZ.monitoring.moveVelocitySelected := FALSE;
   cmSepaGripperAxisZ.monitoring.stopSelected := FALSE;
   cmSepaGripperAxisZ.monitoring.fastStopSelected := FALSE;
   cmSepaGripperAxisZ.monitoring.torqueLimitingSelected := FALSE;
   cmSepaGripperAxisZ.monitoring.homingSelected := FALSE;
   cmSepaGripperAxisZ.monitoring.posRelativeSelected := FALSE;
   cmSepaGripperAxisZ.monitoring.posAbsoluteSelected := FALSE;
   cmSepaGripperAxisZ.monitoring.posSuperimposedSelected := FALSE;
   cmSepaGripperAxisZ.monitoring.haltSuperimposedSelected := FALSE;
   cmSepaGripperAxisZ.monitoring.commandBusy := FALSE;
   cmSepaGripperAxisZ.monitoring.commandDone := FALSE;
   cmSepaGripperAxisZ.monitoring.commandAborted := FALSE;
   cmSepaGripperAxisZ.monitoring.homingCommandBusy := FALSE;
   cmSepaGripperAxisZ.monitoring.homingCommandDone := FALSE;
   cmSepaGripperAxisZ.monitoring.homingCommandAborted := FALSE;
   cmSepaGripperAxisZ.monitoring.superimposedBusy := FALSE;
   cmSepaGripperAxisZ.monitoring.superimposedDone := FALSE;
   cmSepaGripperAxisZ.monitoring.superimposedAborted := FALSE;
   cmSepaGripperAxisZ.monitoring.actualPosition := 159.839;
   cmSepaGripperAxisZ.monitoring.actualSpeed := 0.0;
   cmSepaGripperAxisZ.monitoring.speedUnit := 1062;
   cmSepaGripperAxisZ.monitoring.positionUnit := 1013;
   cmSepaGripperAxisZ.monitoring.axisType := 1;
   cmSepaGripperAxisZ.monitoring.interlockGeneralOut := TRUE;
   cmSepaGripperAxisZ.monitoring.interlockJogForwardOut := TRUE;
   cmSepaGripperAxisZ.monitoring.interlockJogBackwardOut := TRUE;
   cmSepaGripperAxisC.commandConfiguration.generalSettings.stopOnError := TRUE;
   cmSepaGripperAxisC.commandConfiguration.generalSettings.resetWithRestart := FALSE;
   cmSepaGripperAxisC.commandConfiguration.generalSettings.abortWaitingSyncCmd := TRUE;
   cmSepaGripperAxisC.commandConfiguration.power.startMode := 1;
   cmSepaGripperAxisC.commandConfiguration.power.stopMode := 0;
   cmSepaGripperAxisC.commandConfiguration.power.syncMotionSimulation := FALSE;
   cmSepaGripperAxisC.commandConfiguration.power.syncMotionSimulationExtendedMode := -1;
   cmSepaGripperAxisC.commandConfiguration.jog.velocity := 0.0;
   cmSepaGripperAxisC.commandConfiguration.jog.acceleration := -1.0;
   cmSepaGripperAxisC.commandConfiguration.jog.deceleration := -1.0;
   cmSepaGripperAxisC.commandConfiguration.jog.jerk := -1.0;
   cmSepaGripperAxisC.commandConfiguration.jog.positionControlled := TRUE;
   cmSepaGripperAxisC.commandConfiguration.jog.increment := 0.0;
   cmSepaGripperAxisC.commandConfiguration.jog.mode := 0;
   cmSepaGripperAxisC.commandConfiguration.moveVelocity.velocity := 0.0;
   cmSepaGripperAxisC.commandConfiguration.moveVelocity.acceleration := -1.0;
   cmSepaGripperAxisC.commandConfiguration.moveVelocity.deceleration := -1.0;
   cmSepaGripperAxisC.commandConfiguration.moveVelocity.jerk := -1.0;
   cmSepaGripperAxisC.commandConfiguration.moveVelocity.direction := 0;
   cmSepaGripperAxisC.commandConfiguration.moveVelocity.positionControlled := TRUE;
   cmSepaGripperAxisC.commandConfiguration.moveVelocity.velocityChangeOnTheFly := FALSE;
   cmSepaGripperAxisC.commandConfiguration.stop.deceleration := -1.0;
   cmSepaGripperAxisC.commandConfiguration.stop.jerk := -1.0;
   cmSepaGripperAxisC.commandConfiguration.stop.abortAcceleration := FALSE;
   cmSepaGripperAxisC.commandConfiguration.fastStop.deceleration := -1.0;
   cmSepaGripperAxisC.commandConfiguration.fastStop.jerk := -1.0;
   cmSepaGripperAxisC.commandConfiguration.fastStop.abortAcceleration := FALSE;
   cmSepaGripperAxisC.commandConfiguration.fastStop.replaceStopPossible := FALSE;
   cmSepaGripperAxisC.commandConfiguration.torqueLimiting.limit := -1.0;
   cmSepaGripperAxisC.commandConfiguration.torqueLimiting.mode := 0;
   cmSepaGripperAxisC.commandConfiguration.homing.position := 0.0;
   cmSepaGripperAxisC.commandConfiguration.homing.mode := 0;
   cmSepaGripperAxisC.commandConfiguration.homing.sensor := 0;
   cmSepaGripperAxisC.commandConfiguration.homing.extendedMode := -1;
   cmSepaGripperAxisC.commandConfiguration.homing.extendedModeTorqueLimit := 0.0;
   cmSepaGripperAxisC.commandConfiguration.homing.extendedModeTargetPosition := 0.0;
   cmSepaGripperAxisC.commandConfiguration.posRelative.distance := 0.0;
   cmSepaGripperAxisC.commandConfiguration.posRelative.velocity := -1.0;
   cmSepaGripperAxisC.commandConfiguration.posRelative.acceleration := -1.0;
   cmSepaGripperAxisC.commandConfiguration.posRelative.deceleration := -1.0;
   cmSepaGripperAxisC.commandConfiguration.posRelative.jerk := -1.0;
   cmSepaGripperAxisC.commandConfiguration.posRelative.direction := 0;
   cmSepaGripperAxisC.commandConfiguration.posAbsolute.position := 0.0;
   cmSepaGripperAxisC.commandConfiguration.posAbsolute.velocity := -1.0;
   cmSepaGripperAxisC.commandConfiguration.posAbsolute.acceleration := -1.0;
   cmSepaGripperAxisC.commandConfiguration.posAbsolute.deceleration := -1.0;
   cmSepaGripperAxisC.commandConfiguration.posAbsolute.jerk := -1.0;
   cmSepaGripperAxisC.commandConfiguration.posAbsolute.direction := 1;
   cmSepaGripperAxisC.commandConfiguration.posAbsolute.positionChangeOnTheFly := FALSE;
   cmSepaGripperAxisC.commandConfiguration.posAbsolute.velocityChangeOnTheFly := FALSE;
   cmSepaGripperAxisC.commandConfiguration.posSuperimposed.distance := 0.0;
   cmSepaGripperAxisC.commandConfiguration.posSuperimposed.velocityDiff := -1.0;
   cmSepaGripperAxisC.commandConfiguration.posSuperimposed.acceleration := -1.0;
   cmSepaGripperAxisC.commandConfiguration.posSuperimposed.deceleration := -1.0;
   cmSepaGripperAxisC.commandConfiguration.posSuperimposed.jerk := -1.0;
   cmSepaGripperAxisC.commandConfiguration.posSuperimposed.direction := 0;
   cmSepaGripperAxisC.commandConfiguration.haltSuperimposed.deceleration := -1.0;
   cmSepaGripperAxisC.commandConfiguration.haltSuperimposed.jerk := -1.0;
   cmSepaGripperAxisC.commandConfiguration.haltSuperimposed.abortAcceleration := FALSE;
   cmSepaGripperAxisC.commandConfiguration.gearInRelative.ratioNumerator := 1;
   cmSepaGripperAxisC.commandConfiguration.gearInRelative.ratioDenominator := 1;
   cmSepaGripperAxisC.commandConfiguration.gearInRelative.acceleration := -1.0;
   cmSepaGripperAxisC.commandConfiguration.gearInRelative.deceleration := -1.0;
   cmSepaGripperAxisC.commandConfiguration.gearInRelative.jerk := -1.0;
   cmSepaGripperAxisC.commandConfiguration.gearInRelative.ratioChangeOnTheFly := FALSE;
   cmSepaGripperAxisC.commandConfiguration.gearInAbsolute.ratioNumerator := 1;
   cmSepaGripperAxisC.commandConfiguration.gearInAbsolute.ratioDenominator := 1;
   cmSepaGripperAxisC.commandConfiguration.gearInAbsolute.masterSyncPosition := 0.0;
   cmSepaGripperAxisC.commandConfiguration.gearInAbsolute.slaveSyncPosition := 0.0;
   cmSepaGripperAxisC.commandConfiguration.gearInAbsolute.syncProfileReference := 1;
   cmSepaGripperAxisC.commandConfiguration.gearInAbsolute.masterStartDistance := 0.0;
   cmSepaGripperAxisC.commandConfiguration.gearInAbsolute.velocity := -1.0;
   cmSepaGripperAxisC.commandConfiguration.gearInAbsolute.acceleration := -1.0;
   cmSepaGripperAxisC.commandConfiguration.gearInAbsolute.deceleration := -1.0;
   cmSepaGripperAxisC.commandConfiguration.gearInAbsolute.jerk := -1.0;
   cmSepaGripperAxisC.commandConfiguration.gearInAbsolute.syncDirection := 1;
   cmSepaGripperAxisC.commandConfiguration.gearInAbsolute.ratioChangeOnTheFly := FALSE;
   cmSepaGripperAxisC.commandConfiguration.gearInVelocity.continuousUpdate := FALSE;
   cmSepaGripperAxisC.commandConfiguration.gearInVelocity.ratioNumerator := 1;
   cmSepaGripperAxisC.commandConfiguration.gearInVelocity.ratioDenominator := 1;
   cmSepaGripperAxisC.commandConfiguration.gearInVelocity.acceleration := -1.0;
   cmSepaGripperAxisC.commandConfiguration.gearInVelocity.deceleration := -1.0;
   cmSepaGripperAxisC.commandConfiguration.gearInVelocity.jerk := -1.0;
   cmSepaGripperAxisC.commandConfiguration.gearInVelocity.positionControlled := FALSE;
   cmSepaGripperAxisC.commandConfiguration.camIn.masterOffset := 0.0;
   cmSepaGripperAxisC.commandConfiguration.camIn.slaveOffset := 0.0;
   cmSepaGripperAxisC.commandConfiguration.camIn.masterScaling := 1.0;
   cmSepaGripperAxisC.commandConfiguration.camIn.slaveScaling := 1.0;
   cmSepaGripperAxisC.commandConfiguration.camIn.masterSyncPosition := 0.0;
   cmSepaGripperAxisC.commandConfiguration.camIn.syncProfileReference := 1;
   cmSepaGripperAxisC.commandConfiguration.camIn.masterStartDistance := 0.0;
   cmSepaGripperAxisC.commandConfiguration.camIn.velocity := -1.0;
   cmSepaGripperAxisC.commandConfiguration.camIn.acceleration := -1.0;
   cmSepaGripperAxisC.commandConfiguration.camIn.deceleration := -1.0;
   cmSepaGripperAxisC.commandConfiguration.camIn.jerk := -1.0;
   cmSepaGripperAxisC.commandConfiguration.camIn.applicationMode := 0;
   cmSepaGripperAxisC.commandConfiguration.camIn.syncDirection := 1;
   cmSepaGripperAxisC.commandConfiguration.gearOutCamOut.slavePosition := 0.0;
   cmSepaGripperAxisC.commandConfiguration.gearOutCamOut.syncProfileReference := 1;
   cmSepaGripperAxisC.commandConfiguration.gearOutCamOut.masterStopDistance := 0.0;
   cmSepaGripperAxisC.commandConfiguration.gearOutCamOut.deceleration := -1.0;
   cmSepaGripperAxisC.commandConfiguration.gearOutCamOut.jerk := -1.0;
   cmSepaGripperAxisC.commandConfiguration.gearOutCamOut.syncOutDirection := 3;
   cmSepaGripperAxisC.commandConfiguration.gearOutCamOut.gearOutCamOutMode := -1;
   cmSepaGripperAxisC.commandConfiguration.phasing.phaseShift := 0.0;
   cmSepaGripperAxisC.commandConfiguration.phasing.velocity := -1.0;
   cmSepaGripperAxisC.commandConfiguration.phasing.acceleration := -1.0;
   cmSepaGripperAxisC.commandConfiguration.phasing.deceleration := -1.0;
   cmSepaGripperAxisC.commandConfiguration.phasing.jerk := -1.0;
   cmSepaGripperAxisC.commandConfiguration.phasing.profileReference := 0;
   cmSepaGripperAxisC.commandConfiguration.phasing.phasingDistance := 0.0;
   cmSepaGripperAxisC.commandConfiguration.phasing.startPosition := 0.0;
   cmSepaGripperAxisC.commandConfiguration.phasing.direction := 3;
   cmSepaGripperAxisC.commandConfiguration.phasing.phaseAbsolute := TRUE;
   cmSepaGripperAxisC.commandConfiguration.phasing.phaseShiftChangeOnTheFly := FALSE;
   cmSepaGripperAxisC.commandConfiguration.offset.offset := 0.0;
   cmSepaGripperAxisC.commandConfiguration.offset.profileReference := 1;
   cmSepaGripperAxisC.commandConfiguration.offset.offsetDistance := 0.0;
   cmSepaGripperAxisC.commandConfiguration.offset.startPosition := 0.0;
   cmSepaGripperAxisC.commandConfiguration.offset.direction := 3;
   cmSepaGripperAxisC.commandConfiguration.offset.offsetAbsolute := TRUE;
   cmSepaGripperAxisC.commandConfiguration.offset.offsetChangeOnTheFly := FALSE;
   cmSepaGripperAxisC.commands.enableAxis := FALSE;
   cmSepaGripperAxisC.commands.resetAxis := FALSE;
   cmSepaGripperAxisC.commands.openBrake := FALSE;
   cmSepaGripperAxisC.commands.jogForward := FALSE;
   cmSepaGripperAxisC.commands.jogBackward := FALSE;
   cmSepaGripperAxisC.commands.moveVelocity := FALSE;
   cmSepaGripperAxisC.commands.stop := FALSE;
   cmSepaGripperAxisC.commands.fastStop := FALSE;
   cmSepaGripperAxisC.commands.torqueLimiting := FALSE;
   cmSepaGripperAxisC.commands.homing := FALSE;
   cmSepaGripperAxisC.commands.posRelative := FALSE;
   cmSepaGripperAxisC.commands.posAbsolute := FALSE;
   cmSepaGripperAxisC.commands.posSuperimposed := FALSE;
   cmSepaGripperAxisC.commands.haltSuperimposed := FALSE;
   cmSepaGripperAxisC.commands.selectSetPosition := -1;
   cmSepaGripperAxisC.commands.reset := FALSE;
   cmJRWinderRearAxisY.commandConfiguration.generalSettings.stopOnError := TRUE;
   cmJRWinderRearAxisY.commandConfiguration.generalSettings.resetWithRestart := FALSE;
   cmJRWinderRearAxisY.commandConfiguration.generalSettings.abortWaitingSyncCmd := TRUE;
   cmJRWinderRearAxisY.commandConfiguration.power.startMode := 1;
   cmJRWinderRearAxisY.commandConfiguration.power.stopMode := 0;
   cmJRWinderRearAxisY.commandConfiguration.power.syncMotionSimulation := FALSE;
   cmJRWinderRearAxisY.commandConfiguration.power.syncMotionSimulationExtendedMode := -1;
   cmJRWinderRearAxisY.commandConfiguration.jog.velocity := 0.0;
   cmJRWinderRearAxisY.commandConfiguration.jog.acceleration := -1.0;
   cmJRWinderRearAxisY.commandConfiguration.jog.deceleration := -1.0;
   cmJRWinderRearAxisY.commandConfiguration.jog.jerk := -1.0;
   cmJRWinderRearAxisY.commandConfiguration.jog.positionControlled := TRUE;
   cmJRWinderRearAxisY.commandConfiguration.jog.increment := 0.0;
   cmJRWinderRearAxisY.commandConfiguration.jog.mode := 0;
   cmJRWinderRearAxisY.commandConfiguration.moveVelocity.velocity := 0.0;
   cmJRWinderRearAxisY.commandConfiguration.moveVelocity.acceleration := -1.0;
   cmJRWinderRearAxisY.commandConfiguration.moveVelocity.deceleration := -1.0;
   cmJRWinderRearAxisY.commandConfiguration.moveVelocity.jerk := -1.0;
   cmJRWinderRearAxisY.commandConfiguration.moveVelocity.direction := 0;
   cmJRWinderRearAxisY.commandConfiguration.moveVelocity.positionControlled := TRUE;
   cmJRWinderRearAxisY.commandConfiguration.moveVelocity.velocityChangeOnTheFly := FALSE;
   cmJRWinderRearAxisY.commandConfiguration.stop.deceleration := -1.0;
   cmJRWinderRearAxisY.commandConfiguration.stop.jerk := -1.0;
   cmJRWinderRearAxisY.commandConfiguration.stop.abortAcceleration := FALSE;
   cmJRWinderRearAxisY.commandConfiguration.fastStop.deceleration := -1.0;
   cmJRWinderRearAxisY.commandConfiguration.fastStop.jerk := -1.0;
   cmJRWinderRearAxisY.commandConfiguration.fastStop.abortAcceleration := FALSE;
   cmJRWinderRearAxisY.commandConfiguration.fastStop.replaceStopPossible := FALSE;
   cmJRWinderRearAxisY.commandConfiguration.torqueLimiting.limit := -1.0;
   cmJRWinderRearAxisY.commandConfiguration.torqueLimiting.mode := 0;
   cmJRWinderRearAxisY.commandConfiguration.homing.position := 0.0;
   cmJRWinderRearAxisY.commandConfiguration.homing.mode := 0;
   cmJRWinderRearAxisY.commandConfiguration.homing.sensor := 0;
   cmJRWinderRearAxisY.commandConfiguration.homing.extendedMode := -1;
   cmJRWinderRearAxisY.commandConfiguration.homing.extendedModeTorqueLimit := 0.0;
   cmJRWinderRearAxisY.commandConfiguration.homing.extendedModeTargetPosition := 0.0;
   cmJRWinderRearAxisY.commandConfiguration.posRelative.distance := 0.0;
   cmJRWinderRearAxisY.commandConfiguration.posRelative.velocity := -1.0;
   cmJRWinderRearAxisY.commandConfiguration.posRelative.acceleration := -1.0;
